LIN {X 39.082,Y -3.308,Z -37.430,A -90.000,B 90.000,C 0.000} C_DIS
LIN {X 39.427,Y -3.308,Z -37.547,A -90.000,B 90.000,C 0.000} C_DIS
LIN {X 39.464,Y -3.308,Z -37.560,A -90.000,B 90.000,C 0.000} C_DIS
LIN {X 41.255,Y -3.308,Z -38.096,A -90.000,B 90.000,C 0.000} C_DIS
LIN {X 41.425,Y -3.308,Z -38.147,A -90.000,B 90.000,C 0.000} C_DIS
LIN {X 41.590,Y -3.308,Z -38.202,A -90.000,B 90.000,C 0.000} C_DIS
LIN {X 41.777,Y -3.308,Z -38.264,A -90.000,B 90.000,C 0.000} C_DIS
LIN {X 42.094,Y -3.308,Z -38.369,A -90.000,B 90.000,C 0.000} C_DIS
LIN {X 42.169,Y -3.308,Z -38.394,A -90.000,B 90.000,C 0.000} C_DIS
LIN {X 42.347,Y -3.308,Z -38.454,A -90.000,B 90.000,C 0.000} C_DIS
LIN {X 42.646,Y -3.308,Z -38.553,A -90.000,B 90.000,C 0.000} C_DIS
LIN {X 43.376,Y -3.308,Z -38.765,A -90.000,B 90.000,C 0.000} C_DIS
LIN {X 43.430,Y -3.308,Z -38.780,A -90.000,B 90.000,C 0.000} C_DIS
LIN {X 43.466,Y -3.308,Z -38.791,A -90.000,B 90.000,C 0.000} C_DIS
LIN {X 43.779,Y -3.308,Z -38.884,A -90.000,B 90.000,C 0.000} C_DIS
LIN {X 43.869,Y -3.308,Z -38.911,A -90.000,B 90.000,C 0.000} C_DIS
LIN {X 43.897,Y -3.308,Z -38.920,A -90.000,B 90.000,C 0.000} C_DIS
LIN {X 44.112,Y -3.308,Z -38.995,A -90.000,B 90.000,C 0.000} C_DIS
LIN {X 45.330,Y -3.308,Z -39.423,A -90.000,B 90.000,C 0.000} C_DIS
LIN {X 46.342,Y -3.308,Z -39.779,A -90.000,B 90.000,C 0.000} C_DIS
LIN {X 46.474,Y -3.308,Z -39.825,A -90.000,B 90.000,C 0.000} C_DIS
LIN {X 46.539,Y -3.308,Z -39.848,A -90.000,B 90.000,C 0.000} C_DIS
LIN {X 46.539,Y -60.000,Z -39.848,A -90.000,B 90.000,C 0.000} C_DIS
LIN {X 103.720,Y -60.000,Z -88.159,A -90.000,B 90.000,C 0.000} C_DIS
LIN {X 103.720,Y -3.308,Z -88.159,A -90.000,B 90.000,C 0.000} C_DIS
LIN {X 103.972,Y -3.308,Z -88.700,A -90.000,B 90.000,C 0.000} C_DIS
LIN {X 104.338,Y -3.308,Z -89.488,A -90.000,B 90.000,C 0.000} C_DIS
LIN {X 104.627,Y -3.308,Z -90.185,A -90.000,B 90.000,C 0.000} C_DIS
LIN {X 104.874,Y -3.308,Z -90.779,A -90.000,B 90.000,C 0.000} C_DIS
LIN {X 104.949,Y -3.308,Z -90.978,A -90.000,B 90.000,C 0.000} C_DIS
LIN {X 105.045,Y -3.308,Z -91.235,A -90.000,B 90.000,C 0.000} C_DIS
LIN {X 105.277,Y -3.308,Z -91.885,A -90.000,B 90.000,C 0.000} C_DIS
LIN {X 105.456,Y -3.308,Z -92.386,A -90.000,B 90.000,C 0.000} C_DIS
LIN {X 105.632,Y -3.308,Z -92.970,A -90.000,B 90.000,C 0.000} C_DIS
LIN {X 105.781,Y -3.308,Z -93.463,A -90.000,B 90.000,C 0.000} C_DIS
LIN {X 105.840,Y -3.308,Z -93.688,A -90.000,B 90.000,C 0.000} C_DIS
LIN {X 105.905,Y -3.308,Z -93.934,A -90.000,B 90.000,C 0.000} C_DIS
LIN {X 106.039,Y -3.308,Z -94.449,A -90.000,B 90.000,C 0.000} C_DIS
LIN {X 106.184,Y -3.308,Z -95.004,A -90.000,B 90.000,C 0.000} C_DIS
LIN {X 106.291,Y -3.308,Z -95.446,A -90.000,B 90.000,C 0.000} C_DIS
LIN {X 106.458,Y -3.308,Z -96.134,A -90.000,B 90.000,C 0.000} C_DIS
LIN {X 106.542,Y -3.308,Z -96.481,A -90.000,B 90.000,C 0.000} C_DIS
LIN {X 106.764,Y -3.308,Z -97.390,A -90.000,B 90.000,C 0.000} C_DIS
LIN {X 106.814,Y -3.308,Z -97.596,A -90.000,B 90.000,C 0.000} C_DIS
LIN {X 107.111,Y -3.308,Z -98.815,A -90.000,B 90.000,C 0.000} C_DIS
LIN {X 107.114,Y -3.308,Z -98.828,A -90.000,B 90.000,C 0.000} C_DIS
LIN {X 107.136,Y -3.308,Z -98.919,A -90.000,B 90.000,C 0.000} C_DIS
LIN {X 107.500,Y -3.308,Z -100.448,A -90.000,B 90.000,C 0.000} C_DIS
LIN {X 107.513,Y -3.308,Z -100.507,A -90.000,B 90.000,C 0.000} C_DIS
LIN {X 107.940,Y -3.308,Z -102.334,A -90.000,B 90.000,C 0.000} C_DIS
LIN {X 108.408,Y -3.308,Z -104.379,A -90.000,B 90.000,C 0.000} C_DIS
LIN {X 108.438,Y -3.308,Z -104.516,A -90.000,B 90.000,C 0.000} C_DIS
LIN {X 108.935,Y -3.308,Z -106.791,A -90.000,B 90.000,C 0.000} C_DIS
LIN {X 108.968,Y -3.308,Z -106.946,A -90.000,B 90.000,C 0.000} C_DIS
LIN {X 109.472,Y -3.308,Z -109.416,A -90.000,B 90.000,C 0.000} C_DIS
LIN {X 109.504,Y -3.308,Z -109.576,A -90.000,B 90.000,C 0.000} C_DIS
LIN {X 109.988,Y -3.308,Z -112.190,A -90.000,B 90.000,C 0.000} C_DIS
LIN {X 110.019,Y -3.308,Z -112.358,A -90.000,B 90.000,C 0.000} C_DIS
LIN {X 110.455,Y -3.308,Z -115.047,A -90.000,B 90.000,C 0.000} C_DIS
LIN {X 110.486,Y -3.308,Z -115.244,A -90.000,B 90.000,C 0.000} C_DIS
LIN {X 110.492,Y -3.308,Z -115.278,A -90.000,B 90.000,C 0.000} C_DIS
LIN {X 110.561,Y -3.308,Z -115.725,A -90.000,B 90.000,C 0.000} C_DIS
LIN {X 110.947,Y -3.308,Z -118.404,A -90.000,B 90.000,C 0.000} C_DIS
LIN {X 110.982,Y -3.308,Z -118.648,A -90.000,B 90.000,C 0.000} C_DIS
LIN {X 111.318,Y -3.308,Z -121.238,A -90.000,B 90.000,C 0.000} C_DIS
LIN {X 111.357,Y -3.308,Z -121.542,A -90.000,B 90.000,C 0.000} C_DIS
LIN {X 111.645,Y -3.308,Z -123.972,A -90.000,B 90.000,C 0.000} C_DIS
LIN {X 111.687,Y -3.308,Z -124.342,A -90.000,B 90.000,C 0.000} C_DIS
LIN {X 111.725,Y -3.308,Z -124.720,A -90.000,B 90.000,C 0.000} C_DIS
LIN {X 111.972,Y -3.308,Z -126.984,A -90.000,B 90.000,C 0.000} C_DIS
LIN {X 112.002,Y -3.308,Z -127.340,A -90.000,B 90.000,C 0.000} C_DIS
LIN {X 112.036,Y -3.308,Z -127.702,A -90.000,B 90.000,C 0.000} C_DIS
LIN {X 112.062,Y -3.308,Z -127.978,A -90.000,B 90.000,C 0.000} C_DIS
LIN {X 112.218,Y -3.308,Z -129.639,A -90.000,B 90.000,C 0.000} C_DIS
LIN {X 112.242,Y -3.308,Z -129.971,A -90.000,B 90.000,C 0.000} C_DIS
LIN {X 112.397,Y -3.308,Z -132.041,A -90.000,B 90.000,C 0.000} C_DIS
LIN {X 112.415,Y -3.308,Z -132.287,A -90.000,B 90.000,C 0.000} C_DIS
LIN {X 112.415,Y -3.308,Z -132.288,A -90.000,B 90.000,C 0.000} C_DIS
LIN {X 112.440,Y -3.308,Z -132.769,A -90.000,B 90.000,C 0.000} C_DIS
LIN {X 112.440,Y -3.308,Z -132.779,A -90.000,B 90.000,C 0.000} C_DIS
LIN {X 112.584,Y -3.308,Z -135.554,A -90.000,B 90.000,C 0.000} C_DIS
LIN {X 112.669,Y -3.308,Z -138.331,A -90.000,B 90.000,C 0.000} C_DIS
LIN {X 112.673,Y -3.308,Z -138.592,A -90.000,B 90.000,C 0.000} C_DIS
LIN {X 112.707,Y -3.308,Z -141.431,A -90.000,B 90.000,C 0.000} C_DIS
LIN {X 112.707,Y -3.308,Z -141.847,A -90.000,B 90.000,C 0.000} C_DIS
LIN {X 112.692,Y -3.308,Z -144.707,A -90.000,B 90.000,C 0.000} C_DIS
LIN {X 112.684,Y -3.308,Z -145.286,A -90.000,B 90.000,C 0.000} C_DIS
LIN {X 112.623,Y -3.308,Z -148.138,A -90.000,B 90.000,C 0.000} C_DIS
LIN {X 112.620,Y -3.308,Z -148.286,A -90.000,B 90.000,C 0.000} C_DIS
LIN {X 112.607,Y -3.308,Z -148.918,A -90.000,B 90.000,C 0.000} C_DIS
LIN {X 112.605,Y -3.308,Z -148.961,A -90.000,B 90.000,C 0.000} C_DIS
LIN {X 112.590,Y -3.308,Z -149.394,A -90.000,B 90.000,C 0.000} C_DIS
LIN {X 112.473,Y -3.308,Z -152.616,A -90.000,B 90.000,C 0.000} C_DIS
LIN {X 112.455,Y -3.308,Z -153.020,A -90.000,B 90.000,C 0.000} C_DIS
LIN {X 112.452,Y -3.308,Z -153.066,A -90.000,B 90.000,C 0.000} C_DIS
LIN {X 112.429,Y -3.308,Z -153.561,A -90.000,B 90.000,C 0.000} C_DIS
LIN {X 112.272,Y -3.308,Z -156.797,A -90.000,B 90.000,C 0.000} C_DIS
LIN {X 112.267,Y -3.308,Z -156.875,A -90.000,B 90.000,C 0.000} C_DIS
LIN {X 112.051,Y -3.308,Z -160.639,A -90.000,B 90.000,C 0.000} C_DIS
LIN {X 112.041,Y -3.308,Z -160.788,A -90.000,B 90.000,C 0.000} C_DIS
LIN {X 111.803,Y -3.308,Z -164.523,A -90.000,B 90.000,C 0.000} C_DIS
LIN {X 111.556,Y -3.308,Z -168.190,A -90.000,B 90.000,C 0.000} C_DIS
LIN {X 111.538,Y -3.308,Z -168.428,A -90.000,B 90.000,C 0.000} C_DIS
LIN {X 111.279,Y -3.308,Z -171.994,A -90.000,B 90.000,C 0.000} C_DIS
LIN {X 111.258,Y -3.308,Z -172.254,A -90.000,B 90.000,C 0.000} C_DIS
LIN {X 110.991,Y -3.308,Z -175.641,A -90.000,B 90.000,C 0.000} C_DIS
LIN {X 110.967,Y -3.308,Z -175.902,A -90.000,B 90.000,C 0.000} C_DIS
LIN {X 110.692,Y -3.308,Z -179.031,A -90.000,B 90.000,C 0.000} C_DIS
LIN {X 110.688,Y -3.308,Z -179.076,A -90.000,B 90.000,C 0.000} C_DIS
LIN {X 110.671,Y -3.308,Z -179.262,A -90.000,B 90.000,C 0.000} C_DIS
LIN {X 110.455,Y -3.308,Z -181.401,A -90.000,B 90.000,C 0.000} C_DIS
LIN {X 110.368,Y -3.308,Z -182.260,A -90.000,B 90.000,C 0.000} C_DIS
LIN {X 110.143,Y -3.308,Z -184.245,A -90.000,B 90.000,C 0.000} C_DIS
LIN {X 110.061,Y -3.308,Z -184.967,A -90.000,B 90.000,C 0.000} C_DIS
LIN {X 109.829,Y -3.308,Z -186.841,A -90.000,B 90.000,C 0.000} C_DIS
LIN {X 109.752,Y -3.308,Z -187.467,A -90.000,B 90.000,C 0.000} C_DIS
LIN {X 109.519,Y -3.308,Z -189.255,A -90.000,B 90.000,C 0.000} C_DIS
LIN {X 109.442,Y -3.308,Z -189.847,A -90.000,B 90.000,C 0.000} C_DIS
LIN {X 109.426,Y -3.308,Z -189.963,A -90.000,B 90.000,C 0.000} C_DIS
LIN {X 109.200,Y -3.308,Z -191.680,A -90.000,B 90.000,C 0.000} C_DIS
LIN {X 109.115,Y -3.308,Z -192.320,A -90.000,B 90.000,C 0.000} C_DIS
LIN {X 108.873,Y -3.308,Z -194.068,A -90.000,B 90.000,C 0.000} C_DIS
LIN {X 108.760,Y -3.308,Z -194.885,A -90.000,B 90.000,C 0.000} C_DIS
LIN {X 108.715,Y -3.308,Z -195.198,A -90.000,B 90.000,C 0.000} C_DIS
LIN {X 108.447,Y -3.308,Z -197.014,A -90.000,B 90.000,C 0.000} C_DIS
LIN {X 108.278,Y -3.308,Z -198.163,A -90.000,B 90.000,C 0.000} C_DIS
LIN {X 107.982,Y -3.308,Z -200.060,A -90.000,B 90.000,C 0.000} C_DIS
LIN {X 107.713,Y -3.308,Z -201.787,A -90.000,B 90.000,C 0.000} C_DIS
LIN {X 107.405,Y -3.308,Z -203.667,A -90.000,B 90.000,C 0.000} C_DIS
LIN {X 106.975,Y -3.308,Z -206.301,A -90.000,B 90.000,C 0.000} C_DIS
LIN {X 106.701,Y -3.308,Z -207.830,A -90.000,B 90.000,C 0.000} C_DIS
LIN {X 106.050,Y -3.308,Z -211.464,A -90.000,B 90.000,C 0.000} C_DIS
LIN {X 105.858,Y -3.308,Z -212.410,A -90.000,B 90.000,C 0.000} C_DIS
LIN {X 104.921,Y -3.308,Z -217.034,A -90.000,B 90.000,C 0.000} C_DIS
LIN {X 104.861,Y -3.308,Z -217.290,A -90.000,B 90.000,C 0.000} C_DIS
LIN {X 104.401,Y -3.308,Z -219.248,A -90.000,B 90.000,C 0.000} C_DIS
LIN {X 103.570,Y -3.308,Z -222.773,A -90.000,B 90.000,C 0.000} C_DIS
LIN {X 103.568,Y -3.308,Z -222.782,A -90.000,B 90.000,C 0.000} C_DIS
LIN {X 103.460,Y -3.308,Z -223.227,A -90.000,B 90.000,C 0.000} C_DIS
LIN {X 103.428,Y -3.308,Z -223.346,A -90.000,B 90.000,C 0.000} C_DIS
LIN {X 101.875,Y -3.308,Z -228.890,A -90.000,B 90.000,C 0.000} C_DIS
LIN {X 101.788,Y -3.308,Z -229.169,A -90.000,B 90.000,C 0.000} C_DIS
LIN {X 100.060,Y -3.308,Z -234.610,A -90.000,B 90.000,C 0.000} C_DIS
LIN {X 99.904,Y -3.308,Z -235.072,A -90.000,B 90.000,C 0.000} C_DIS
LIN {X 99.844,Y -3.308,Z -235.247,A -90.000,B 90.000,C 0.000} C_DIS
LIN {X 99.341,Y -3.308,Z -236.708,A -90.000,B 90.000,C 0.000} C_DIS
LIN {X 98.008,Y -3.308,Z -240.566,A -90.000,B 90.000,C 0.000} C_DIS
LIN {X 97.126,Y -3.308,Z -243.023,A -90.000,B 90.000,C 0.000} C_DIS
LIN {X 96.931,Y -3.308,Z -243.561,A -90.000,B 90.000,C 0.000} C_DIS
LIN {X 96.931,Y -60.000,Z -243.561,A -90.000,B 90.000,C 0.000} C_DIS
LIN {X 103.942,Y -60.000,Z -88.551,A -90.000,B 90.000,C 0.000} C_DIS
LIN {X 103.942,Y -1.308,Z -88.551,A -90.000,B 90.000,C 0.000} C_DIS
LIN {X 104.175,Y -1.308,Z -89.077,A -90.000,B 90.000,C 0.000} C_DIS
LIN {X 104.366,Y -1.308,Z -89.489,A -90.000,B 90.000,C 0.000} C_DIS
LIN {X 104.694,Y -1.308,Z -90.316,A -90.000,B 90.000,C 0.000} C_DIS
LIN {X 104.887,Y -1.308,Z -90.782,A -90.000,B 90.000,C 0.000} C_DIS
LIN {X 105.061,Y -1.308,Z -91.248,A -90.000,B 90.000,C 0.000} C_DIS
LIN {X 105.471,Y -1.308,Z -92.397,A -90.000,B 90.000,C 0.000} C_DIS
LIN {X 105.797,Y -1.308,Z -93.474,A -90.000,B 90.000,C 0.000} C_DIS
LIN {X 106.202,Y -1.308,Z -95.016,A -90.000,B 90.000,C 0.000} C_DIS
LIN {X 106.649,Y -1.308,Z -96.839,A -90.000,B 90.000,C 0.000} C_DIS
LIN {X 107.139,Y -1.308,Z -98.829,A -90.000,B 90.000,C 0.000} C_DIS
LIN {X 107.348,Y -1.308,Z -99.694,A -90.000,B 90.000,C 0.000} C_DIS
LIN {X 107.535,Y -1.308,Z -100.466,A -90.000,B 90.000,C 0.000} C_DIS
LIN {X 107.981,Y -1.308,Z -102.357,A -90.000,B 90.000,C 0.000} C_DIS
LIN {X 108.482,Y -1.308,Z -104.543,A -90.000,B 90.000,C 0.000} C_DIS
LIN {X 108.811,Y -1.308,Z -106.031,A -90.000,B 90.000,C 0.000} C_DIS
LIN {X 109.029,Y -1.308,Z -107.030,A -90.000,B 90.000,C 0.000} C_DIS
LIN {X 109.354,Y -1.308,Z -108.598,A -90.000,B 90.000,C 0.000} C_DIS
LIN {X 109.573,Y -1.308,Z -109.674,A -90.000,B 90.000,C 0.000} C_DIS
LIN {X 109.886,Y -1.308,Z -111.341,A -90.000,B 90.000,C 0.000} C_DIS
LIN {X 110.096,Y -1.308,Z -112.473,A -90.000,B 90.000,C 0.000} C_DIS
LIN {X 110.570,Y -1.308,Z -115.379,A -90.000,B 90.000,C 0.000} C_DIS
LIN {X 110.644,Y -1.308,Z -115.861,A -90.000,B 90.000,C 0.000} C_DIS
LIN {X 111.073,Y -1.308,Z -118.807,A -90.000,B 90.000,C 0.000} C_DIS
LIN {X 111.459,Y -1.308,Z -121.724,A -90.000,B 90.000,C 0.000} C_DIS
LIN {X 111.654,Y -1.308,Z -123.293,A -90.000,B 90.000,C 0.000} C_DIS
LIN {X 111.804,Y -1.308,Z -124.546,A -90.000,B 90.000,C 0.000} C_DIS
LIN {X 111.944,Y -1.308,Z -125.792,A -90.000,B 90.000,C 0.000} C_DIS
LIN {X 112.113,Y -1.308,Z -127.205,A -90.000,B 90.000,C 0.000} C_DIS
LIN {X 112.238,Y -1.308,Z -128.493,A -90.000,B 90.000,C 0.000} C_DIS
LIN {X 112.386,Y -1.308,Z -129.880,A -90.000,B 90.000,C 0.000} C_DIS
LIN {X 112.447,Y -1.308,Z -130.676,A -90.000,B 90.000,C 0.000} C_DIS
LIN {X 112.614,Y -1.308,Z -132.524,A -90.000,B 90.000,C 0.000} C_DIS
LIN {X 112.665,Y -1.308,Z -133.450,A -90.000,B 90.000,C 0.000} C_DIS
LIN {X 112.792,Y -1.308,Z -135.313,A -90.000,B 90.000,C 0.000} C_DIS
LIN {X 112.817,Y -1.308,Z -135.799,A -90.000,B 90.000,C 0.000} C_DIS
LIN {X 112.906,Y -1.308,Z -137.712,A -90.000,B 90.000,C 0.000} C_DIS
LIN {X 112.943,Y -1.308,Z -138.836,A -90.000,B 90.000,C 0.000} C_DIS
LIN {X 112.993,Y -1.308,Z -140.776,A -90.000,B 90.000,C 0.000} C_DIS
LIN {X 113.012,Y -1.308,Z -142.085,A -90.000,B 90.000,C 0.000} C_DIS
LIN {X 113.024,Y -1.308,Z -144.018,A -90.000,B 90.000,C 0.000} C_DIS
LIN {X 113.019,Y -1.308,Z -145.583,A -90.000,B 90.000,C 0.000} C_DIS
LIN {X 112.990,Y -1.308,Z -147.783,A -90.000,B 90.000,C 0.000} C_DIS
LIN {X 112.966,Y -1.308,Z -149.138,A -90.000,B 90.000,C 0.000} C_DIS
LIN {X 112.932,Y -1.308,Z -150.098,A -90.000,B 90.000,C 0.000} C_DIS
LIN {X 112.836,Y -1.308,Z -153.117,A -90.000,B 90.000,C 0.000} C_DIS
LIN {X 112.787,Y -1.308,Z -154.172,A -90.000,B 90.000,C 0.000} C_DIS
LIN {X 112.665,Y -1.308,Z -156.858,A -90.000,B 90.000,C 0.000} C_DIS
LIN {X 112.602,Y -1.308,Z -157.990,A -90.000,B 90.000,C 0.000} C_DIS
LIN {X 112.456,Y -1.308,Z -160.667,A -90.000,B 90.000,C 0.000} C_DIS
LIN {X 112.381,Y -1.308,Z -161.858,A -90.000,B 90.000,C 0.000} C_DIS
LIN {X 112.222,Y -1.308,Z -164.528,A -90.000,B 90.000,C 0.000} C_DIS
LIN {X 112.060,Y -1.308,Z -167.189,A -90.000,B 90.000,C 0.000} C_DIS
LIN {X 111.977,Y -1.308,Z -168.425,A -90.000,B 90.000,C 0.000} C_DIS
LIN {X 111.811,Y -1.308,Z -171.020,A -90.000,B 90.000,C 0.000} C_DIS
LIN {X 111.722,Y -1.308,Z -172.253,A -90.000,B 90.000,C 0.000} C_DIS
LIN {X 111.551,Y -1.308,Z -174.718,A -90.000,B 90.000,C 0.000} C_DIS
LIN {X 111.281,Y -1.308,Z -178.178,A -90.000,B 90.000,C 0.000} C_DIS
LIN {X 111.184,Y -1.308,Z -179.276,A -90.000,B 90.000,C 0.000} C_DIS
LIN {X 111.000,Y -1.308,Z -181.292,A -90.000,B 90.000,C 0.000} C_DIS
LIN {X 110.891,Y -1.308,Z -182.370,A -90.000,B 90.000,C 0.000} C_DIS
LIN {X 110.637,Y -1.308,Z -184.806,A -90.000,B 90.000,C 0.000} C_DIS
LIN {X 110.351,Y -1.308,Z -187.300,A -90.000,B 90.000,C 0.000} C_DIS
LIN {X 110.065,Y -1.308,Z -189.655,A -90.000,B 90.000,C 0.000} C_DIS
LIN {X 110.039,Y -1.308,Z -189.862,A -90.000,B 90.000,C 0.000} C_DIS
LIN {X 109.783,Y -1.308,Z -191.958,A -90.000,B 90.000,C 0.000} C_DIS
LIN {X 109.461,Y -1.308,Z -194.432,A -90.000,B 90.000,C 0.000} C_DIS
LIN {X 108.986,Y -1.308,Z -197.778,A -90.000,B 90.000,C 0.000} C_DIS
LIN {X 108.937,Y -1.308,Z -198.114,A -90.000,B 90.000,C 0.000} C_DIS
LIN {X 108.377,Y -1.308,Z -201.749,A -90.000,B 90.000,C 0.000} C_DIS
LIN {X 107.631,Y -1.308,Z -206.299,A -90.000,B 90.000,C 0.000} C_DIS
LIN {X 107.482,Y -1.308,Z -207.134,A -90.000,B 90.000,C 0.000} C_DIS
LIN {X 106.688,Y -1.308,Z -211.510,A -90.000,B 90.000,C 0.000} C_DIS
LIN {X 106.478,Y -1.308,Z -212.555,A -90.000,B 90.000,C 0.000} C_DIS
LIN {X 105.535,Y -1.308,Z -217.130,A -90.000,B 90.000,C 0.000} C_DIS
LIN {X 105.249,Y -1.308,Z -218.352,A -90.000,B 90.000,C 0.000} C_DIS
LIN {X 104.157,Y -1.308,Z -222.909,A -90.000,B 90.000,C 0.000} C_DIS
LIN {X 104.041,Y -1.308,Z -223.370,A -90.000,B 90.000,C 0.000} C_DIS
LIN {X 103.553,Y -1.308,Z -225.114,A -90.000,B 90.000,C 0.000} C_DIS
LIN {X 103.299,Y -1.308,Z -226.019,A -90.000,B 90.000,C 0.000} C_DIS
LIN {X 102.457,Y -1.308,Z -228.965,A -90.000,B 90.000,C 0.000} C_DIS
LIN {X 101.545,Y -1.308,Z -231.849,A -90.000,B 90.000,C 0.000} C_DIS
LIN {X 100.624,Y -1.308,Z -234.696,A -90.000,B 90.000,C 0.000} C_DIS
LIN {X 100.468,Y -1.308,Z -235.153,A -90.000,B 90.000,C 0.000} C_DIS
LIN {X 99.390,Y -1.308,Z -238.286,A -90.000,B 90.000,C 0.000} C_DIS
LIN {X 98.415,Y -1.308,Z -241.076,A -90.000,B 90.000,C 0.000} C_DIS
LIN {X 97.517,Y -1.308,Z -243.561,A -90.000,B 90.000,C 0.000} C_DIS
LIN {X 97.589,Y -0.997,Z -243.561,A -90.000,B 90.000,C 0.000} C_DIS
LIN {X 97.753,Y -0.254,Z -243.561,A -90.000,B 90.000,C 0.000} C_DIS
LIN {X 97.794,Y -0.012,Z -243.561,A -90.000,B 90.000,C 0.000} C_DIS
LIN {X 98.717,Y -0.012,Z -241.018,A -90.000,B 90.000,C 0.000} C_DIS
LIN {X 100.794,Y -0.012,Z -235.068,A -90.000,B 90.000,C 0.000} C_DIS
LIN {X 100.850,Y -0.012,Z -234.903,A -90.000,B 90.000,C 0.000} C_DIS
LIN {X 102.698,Y -0.012,Z -229.178,A -90.000,B 90.000,C 0.000} C_DIS
LIN {X 104.377,Y -0.012,Z -223.284,A -90.000,B 90.000,C 0.000} C_DIS
LIN {X 104.419,Y -0.012,Z -223.135,A -90.000,B 90.000,C 0.000} C_DIS
LIN {X 105.820,Y -0.012,Z -217.262,A -90.000,B 90.000,C 0.000} C_DIS
LIN {X 106.103,Y -0.012,Z -215.906,A -90.000,B 90.000,C 0.000} C_DIS
LIN {X 107.024,Y -0.012,Z -211.415,A -90.000,B 90.000,C 0.000} C_DIS
LIN {X 107.238,Y -0.012,Z -210.247,A -90.000,B 90.000,C 0.000} C_DIS
LIN {X 107.970,Y -0.012,Z -206.189,A -90.000,B 90.000,C 0.000} C_DIS
LIN {X 108.152,Y -0.012,Z -205.081,A -90.000,B 90.000,C 0.000} C_DIS
LIN {X 108.714,Y -0.012,Z -201.630,A -90.000,B 90.000,C 0.000} C_DIS
LIN {X 109.268,Y -0.012,Z -197.995,A -90.000,B 90.000,C 0.000} C_DIS
LIN {X 109.567,Y -0.012,Z -195.870,A -90.000,B 90.000,C 0.000} C_DIS
LIN {X 109.681,Y -0.012,Z -195.046,A -90.000,B 90.000,C 0.000} C_DIS
LIN {X 109.912,Y -0.012,Z -193.259,A -90.000,B 90.000,C 0.000} C_DIS
LIN {X 110.256,Y -0.012,Z -190.433,A -90.000,B 90.000,C 0.000} C_DIS
LIN {X 110.329,Y -0.012,Z -189.794,A -90.000,B 90.000,C 0.000} C_DIS
LIN {X 110.584,Y -0.012,Z -187.672,A -90.000,B 90.000,C 0.000} C_DIS
LIN {X 110.866,Y -0.012,Z -185.210,A -90.000,B 90.000,C 0.000} C_DIS
LIN {X 111.127,Y -0.012,Z -182.715,A -90.000,B 90.000,C 0.000} C_DIS
LIN {X 111.399,Y -0.012,Z -179.749,A -90.000,B 90.000,C 0.000} C_DIS
LIN {X 111.661,Y -0.012,Z -176.403,A -90.000,B 90.000,C 0.000} C_DIS
LIN {X 111.946,Y -0.012,Z -172.287,A -90.000,B 90.000,C 0.000} C_DIS
LIN {X 112.188,Y -0.012,Z -168.484,A -90.000,B 90.000,C 0.000} C_DIS
LIN {X 112.438,Y -0.012,Z -164.328,A -90.000,B 90.000,C 0.000} C_DIS
LIN {X 112.665,Y -0.012,Z -160.479,A -90.000,B 90.000,C 0.000} C_DIS
LIN {X 112.870,Y -0.012,Z -156.686,A -90.000,B 90.000,C 0.000} C_DIS
LIN {X 113.036,Y -0.012,Z -152.962,A -90.000,B 90.000,C 0.000} C_DIS
LIN {X 113.146,Y -0.012,Z -149.320,A -90.000,B 90.000,C 0.000} C_DIS
LIN {X 113.182,Y -0.012,Z -146.203,A -90.000,B 90.000,C 0.000} C_DIS
LIN {X 113.185,Y -0.012,Z -145.696,A -90.000,B 90.000,C 0.000} C_DIS
LIN {X 113.163,Y -0.012,Z -142.850,A -90.000,B 90.000,C 0.000} C_DIS
LIN {X 113.155,Y -0.012,Z -142.278,A -90.000,B 90.000,C 0.000} C_DIS
LIN {X 113.081,Y -0.012,Z -139.539,A -90.000,B 90.000,C 0.000} C_DIS
LIN {X 113.064,Y -0.012,Z -138.972,A -90.000,B 90.000,C 0.000} C_DIS
LIN {X 112.922,Y -0.012,Z -135.965,A -90.000,B 90.000,C 0.000} C_DIS
LIN {X 112.892,Y -0.012,Z -135.399,A -90.000,B 90.000,C 0.000} C_DIS
LIN {X 112.699,Y -0.012,Z -132.647,A -90.000,B 90.000,C 0.000} C_DIS
LIN {X 112.454,Y -0.012,Z -129.979,A -90.000,B 90.000,C 0.000} C_DIS
LIN {X 112.169,Y -0.012,Z -127.364,A -90.000,B 90.000,C 0.000} C_DIS
LIN {X 111.849,Y -0.012,Z -124.692,A -90.000,B 90.000,C 0.000} C_DIS
LIN {X 111.494,Y -0.012,Z -121.847,A -90.000,B 90.000,C 0.000} C_DIS
LIN {X 111.104,Y -0.012,Z -118.911,A -90.000,B 90.000,C 0.000} C_DIS
LIN {X 110.672,Y -0.012,Z -115.948,A -90.000,B 90.000,C 0.000} C_DIS
LIN {X 110.597,Y -0.012,Z -115.467,A -90.000,B 90.000,C 0.000} C_DIS
LIN {X 110.120,Y -0.012,Z -112.547,A -90.000,B 90.000,C 0.000} C_DIS
LIN {X 109.594,Y -0.012,Z -109.738,A -90.000,B 90.000,C 0.000} C_DIS
LIN {X 109.044,Y -0.012,Z -107.086,A -90.000,B 90.000,C 0.000} C_DIS
LIN {X 108.477,Y -0.012,Z -104.519,A -90.000,B 90.000,C 0.000} C_DIS
LIN {X 107.976,Y -0.012,Z -102.336,A -90.000,B 90.000,C 0.000} C_DIS
LIN {X 107.530,Y -0.012,Z -100.448,A -90.000,B 90.000,C 0.000} C_DIS
LIN {X 107.135,Y -0.012,Z -98.812,A -90.000,B 90.000,C 0.000} C_DIS
LIN {X 106.475,Y -0.012,Z -96.132,A -90.000,B 90.000,C 0.000} C_DIS
LIN {X 106.196,Y -0.012,Z -94.993,A -90.000,B 90.000,C 0.000} C_DIS
LIN {X 105.793,Y -0.012,Z -93.461,A -90.000,B 90.000,C 0.000} C_DIS
LIN {X 105.467,Y -0.012,Z -92.384,A -90.000,B 90.000,C 0.000} C_DIS
LIN {X 105.056,Y -0.012,Z -91.234,A -90.000,B 90.000,C 0.000} C_DIS
LIN {X 104.885,Y -0.012,Z -90.777,A -90.000,B 90.000,C 0.000} C_DIS
LIN {X 104.827,Y -0.012,Z -90.638,A -90.000,B 90.000,C 0.000} C_DIS
LIN {X 104.372,Y -0.012,Z -89.491,A -90.000,B 90.000,C 0.000} C_DIS
LIN {X 104.045,Y -0.012,Z -88.752,A -90.000,B 90.000,C 0.000} C_DIS
LIN {X 104.045,Y -60.000,Z -88.752,A -90.000,B 90.000,C 0.000} C_DIS
LIN {X 43.020,Y -60.000,Z -37.966,A -90.000,B 90.000,C 0.000} C_DIS
LIN {X 43.020,Y -0.012,Z -37.966,A -90.000,B 90.000,C 0.000} C_DIS
LIN {X 42.676,Y -0.012,Z -37.859,A -90.000,B 90.000,C 0.000} C_DIS
LIN {X 39.938,Y -0.012,Z -37.046,A -90.000,B 90.000,C 0.000} C_DIS
LIN {X 39.474,Y -0.012,Z -36.914,A -90.000,B 90.000,C 0.000} C_DIS
LIN {X 38.817,Y -0.012,Z -36.731,A -90.000,B 90.000,C 0.000} C_DIS
LIN {X 36.912,Y -0.012,Z -36.186,A -90.000,B 90.000,C 0.000} C_DIS
LIN {X 36.067,Y -0.012,Z -35.963,A -90.000,B 90.000,C 0.000} C_DIS
LIN {X 34.152,Y -0.012,Z -35.416,A -90.000,B 90.000,C 0.000} C_DIS
LIN {X 32.390,Y -0.012,Z -34.936,A -90.000,B 90.000,C 0.000} C_DIS
LIN {X 32.190,Y -0.012,Z -34.876,A -90.000,B 90.000,C 0.000} C_DIS
LIN {X 30.670,Y -0.012,Z -34.493,A -90.000,B 90.000,C 0.000} C_DIS
LIN {X 30.375,Y -0.012,Z -34.410,A -90.000,B 90.000,C 0.000} C_DIS
LIN {X 29.074,Y -0.012,Z -34.123,A -90.000,B 90.000,C 0.000} C_DIS
LIN {X 28.686,Y -0.012,Z -34.028,A -90.000,B 90.000,C 0.000} C_DIS
LIN {X 28.208,Y -0.012,Z -33.939,A -90.000,B 90.000,C 0.000} C_DIS
LIN {X 27.702,Y -0.012,Z -33.849,A -90.000,B 90.000,C 0.000} C_DIS
LIN {X 26.733,Y -0.012,Z -33.598,A -90.000,B 90.000,C 0.000} C_DIS
LIN {X 25.280,Y -0.012,Z -33.266,A -90.000,B 90.000,C 0.000} C_DIS
LIN {X 23.854,Y -0.012,Z -32.973,A -90.000,B 90.000,C 0.000} C_DIS
LIN {X 20.821,Y -0.012,Z -32.391,A -90.000,B 90.000,C 0.000} C_DIS
LIN {X 19.125,Y -0.012,Z -32.043,A -90.000,B 90.000,C 0.000} C_DIS
LIN {X 15.767,Y -0.012,Z -31.256,A -90.000,B 90.000,C 0.000} C_DIS
LIN {X 14.185,Y -0.012,Z -30.896,A -90.000,B 90.000,C 0.000} C_DIS
LIN {X 12.581,Y -0.012,Z -30.540,A -90.000,B 90.000,C 0.000} C_DIS
LIN {X 10.880,Y -0.012,Z -30.117,A -90.000,B 90.000,C 0.000} C_DIS
LIN {X 8.865,Y -0.012,Z -29.622,A -90.000,B 90.000,C 0.000} C_DIS
LIN {X 3.891,Y -0.012,Z -28.465,A -90.000,B 90.000,C 0.000} C_DIS
LIN {X 1.041,Y -0.012,Z -27.770,A -90.000,B 90.000,C 0.000} C_DIS
LIN {X -1.976,Y -0.012,Z -26.974,A -90.000,B 90.000,C 0.000} C_DIS
LIN {X -4.624,Y -0.012,Z -26.193,A -90.000,B 90.000,C 0.000} C_DIS
LIN {X -7.412,Y -0.012,Z -25.311,A -90.000,B 90.000,C 0.000} C_DIS
LIN {X -7.754,Y -0.012,Z -25.207,A -90.000,B 90.000,C 0.000} C_DIS
LIN {X -10.062,Y -0.012,Z -24.467,A -90.000,B 90.000,C 0.000} C_DIS
LIN {X -10.863,Y -0.012,Z -24.217,A -90.000,B 90.000,C 0.000} C_DIS
LIN {X -13.621,Y -0.012,Z -23.346,A -90.000,B 90.000,C 0.000} C_DIS
LIN {X -13.820,Y -0.012,Z -23.285,A -90.000,B 90.000,C 0.000} C_DIS
LIN {X -16.774,Y -0.012,Z -22.405,A -90.000,B 90.000,C 0.000} C_DIS
LIN {X -16.893,Y -0.012,Z -22.370,A -90.000,B 90.000,C 0.000} C_DIS
LIN {X -17.636,Y -0.012,Z -22.162,A -90.000,B 90.000,C 0.000} C_DIS
LIN {X -19.279,Y -0.012,Z -21.696,A -90.000,B 90.000,C 0.000} C_DIS
LIN {X -21.539,Y -0.012,Z -21.084,A -90.000,B 90.000,C 0.000} C_DIS
LIN {X -26.043,Y -0.012,Z -19.895,A -90.000,B 90.000,C 0.000} C_DIS
LIN {X -26.588,Y -0.012,Z -19.760,A -90.000,B 90.000,C 0.000} C_DIS
LIN {X -28.502,Y -0.012,Z -19.295,A -90.000,B 90.000,C 0.000} C_DIS
LIN {X -31.206,Y -0.012,Z -18.708,A -90.000,B 90.000,C 0.000} C_DIS
LIN {X -33.757,Y -0.012,Z -18.236,A -90.000,B 90.000,C 0.000} C_DIS
LIN {X -34.712,Y -0.012,Z -18.067,A -90.000,B 90.000,C 0.000} C_DIS
LIN {X -37.747,Y -0.012,Z -17.621,A -90.000,B 90.000,C 0.000} C_DIS
LIN {X -38.152,Y -0.012,Z -17.555,A -90.000,B 90.000,C 0.000} C_DIS
LIN {X -40.937,Y -0.012,Z -17.179,A -90.000,B 90.000,C 0.000} C_DIS
LIN {X -41.696,Y -0.012,Z -17.061,A -90.000,B 90.000,C 0.000} C_DIS
LIN {X -42.842,Y -0.012,Z -16.906,A -90.000,B 90.000,C 0.000} C_DIS
LIN {X -45.181,Y -0.012,Z -16.537,A -90.000,B 90.000,C 0.000} C_DIS
LIN {X -45.737,Y -0.012,Z -16.454,A -90.000,B 90.000,C 0.000} C_DIS
LIN {X -48.058,Y -0.012,Z -16.058,A -90.000,B 90.000,C 0.000} C_DIS
LIN {X -49.516,Y -0.012,Z -15.762,A -90.000,B 90.000,C 0.000} C_DIS
LIN {X -50.309,Y -0.012,Z -15.602,A -90.000,B 90.000,C 0.000} C_DIS
LIN {X -52.298,Y -0.012,Z -15.130,A -90.000,B 90.000,C 0.000} C_DIS
LIN {X -53.891,Y -0.012,Z -14.701,A -90.000,B 90.000,C 0.000} C_DIS
LIN {X -55.198,Y -0.012,Z -14.324,A -90.000,B 90.000,C 0.000} C_DIS
LIN {X -56.332,Y -0.012,Z -14.007,A -90.000,B 90.000,C 0.000} C_DIS
LIN {X -57.641,Y -0.012,Z -13.652,A -90.000,B 90.000,C 0.000} C_DIS
LIN {X -59.127,Y -0.012,Z -13.251,A -90.000,B 90.000,C 0.000} C_DIS
LIN {X -60.166,Y -0.012,Z -12.960,A -90.000,B 90.000,C 0.000} C_DIS
LIN {X -61.184,Y -0.012,Z -12.702,A -90.000,B 90.000,C 0.000} C_DIS
LIN {X -62.291,Y -0.012,Z -12.477,A -90.000,B 90.000,C 0.000} C_DIS
LIN {X -62.770,Y -0.012,Z -12.387,A -90.000,B 90.000,C 0.000} C_DIS
LIN {X -63.035,Y -0.012,Z -12.350,A -90.000,B 90.000,C 0.000} C_DIS
LIN {X -64.074,Y -0.012,Z -12.192,A -90.000,B 90.000,C 0.000} C_DIS
LIN {X -64.556,Y -0.012,Z -12.151,A -90.000,B 90.000,C 0.000} C_DIS
LIN {X -65.927,Y -0.012,Z -12.042,A -90.000,B 90.000,C 0.000} C_DIS
LIN {X -67.369,Y -0.012,Z -11.981,A -90.000,B 90.000,C 0.000} C_DIS
LIN {X -68.812,Y -0.012,Z -11.939,A -90.000,B 90.000,C 0.000} C_DIS
LIN {X -70.189,Y -0.012,Z -11.883,A -90.000,B 90.000,C 0.000} C_DIS
LIN {X -71.023,Y -0.012,Z -11.818,A -90.000,B 90.000,C 0.000} C_DIS
LIN {X -72.129,Y -0.012,Z -11.687,A -90.000,B 90.000,C 0.000} C_DIS
LIN {X -73.241,Y -0.012,Z -11.518,A -90.000,B 90.000,C 0.000} C_DIS
LIN {X -74.294,Y -0.012,Z -11.380,A -90.000,B 90.000,C 0.000} C_DIS
LIN {X -74.779,Y -0.012,Z -11.338,A -90.000,B 90.000,C 0.000} C_DIS
LIN {X -75.788,Y -0.012,Z -11.262,A -90.000,B 90.000,C 0.000} C_DIS
LIN {X -76.595,Y -0.012,Z -11.236,A -90.000,B 90.000,C 0.000} C_DIS
LIN {X -76.881,Y -0.012,Z -11.223,A -90.000,B 90.000,C 0.000} C_DIS
LIN {X -77.658,Y -0.012,Z -11.218,A -90.000,B 90.000,C 0.000} C_DIS
LIN {X -77.953,Y -0.012,Z -11.212,A -90.000,B 90.000,C 0.000} C_DIS
LIN {X -78.827,Y -0.012,Z -11.211,A -90.000,B 90.000,C 0.000} C_DIS
LIN {X -79.219,Y -0.012,Z -11.205,A -90.000,B 90.000,C 0.000} C_DIS
LIN {X -80.206,Y -0.012,Z -11.169,A -90.000,B 90.000,C 0.000} C_DIS
LIN {X -80.638,Y -0.012,Z -11.166,A -90.000,B 90.000,C 0.000} C_DIS
LIN {X -81.548,Y -0.012,Z -11.134,A -90.000,B 90.000,C 0.000} C_DIS
LIN {X -82.119,Y -0.012,Z -11.133,A -90.000,B 90.000,C 0.000} C_DIS
LIN {X -82.935,Y -0.012,Z -11.120,A -90.000,B 90.000,C 0.000} C_DIS
LIN {X -83.757,Y -0.012,Z -11.111,A -90.000,B 90.000,C 0.000} C_DIS
LIN {X -85.248,Y -0.012,Z -11.141,A -90.000,B 90.000,C 0.000} C_DIS
LIN {X -85.753,Y -0.012,Z -11.159,A -90.000,B 90.000,C 0.000} C_DIS
LIN {X -87.138,Y -0.012,Z -11.278,A -90.000,B 90.000,C 0.000} C_DIS
LIN {X -87.533,Y -0.012,Z -11.333,A -90.000,B 90.000,C 0.000} C_DIS
LIN {X -88.765,Y -0.012,Z -11.522,A -90.000,B 90.000,C 0.000} C_DIS
LIN {X -88.932,Y -0.012,Z -11.549,A -90.000,B 90.000,C 0.000} C_DIS
LIN {X -90.192,Y -0.012,Z -11.831,A -90.000,B 90.000,C 0.000} C_DIS
LIN {X -90.405,Y -0.012,Z -11.883,A -90.000,B 90.000,C 0.000} C_DIS
LIN {X -90.656,Y -0.012,Z -11.951,A -90.000,B 90.000,C 0.000} C_DIS
LIN {X -91.880,Y -0.012,Z -12.313,A -90.000,B 90.000,C 0.000} C_DIS
LIN {X -93.124,Y -0.012,Z -12.761,A -90.000,B 90.000,C 0.000} C_DIS
LIN {X -93.538,Y -0.012,Z -12.922,A -90.000,B 90.000,C 0.000} C_DIS
LIN {X -93.992,Y -0.012,Z -13.111,A -90.000,B 90.000,C 0.000} C_DIS
LIN {X -94.547,Y -0.012,Z -13.336,A -90.000,B 90.000,C 0.000} C_DIS
LIN {X -94.813,Y -0.012,Z -13.457,A -90.000,B 90.000,C 0.000} C_DIS
LIN {X -95.652,Y -0.012,Z -13.832,A -90.000,B 90.000,C 0.000} C_DIS
LIN {X -96.130,Y -0.012,Z -14.062,A -90.000,B 90.000,C 0.000} C_DIS
LIN {X -97.061,Y -0.012,Z -14.512,A -90.000,B 90.000,C 0.000} C_DIS
LIN {X -98.451,Y -0.012,Z -15.222,A -90.000,B 90.000,C 0.000} C_DIS
LIN {X -99.427,Y -0.012,Z -15.739,A -90.000,B 90.000,C 0.000} C_DIS
LIN {X -100.226,Y -0.012,Z -16.182,A -90.000,B 90.000,C 0.000} C_DIS
LIN {X -100.368,Y -0.012,Z -16.265,A -90.000,B 90.000,C 0.000} C_DIS
LIN {X -100.488,Y -0.012,Z -16.339,A -90.000,B 90.000,C 0.000} C_DIS
LIN {X -100.938,Y -0.012,Z -16.608,A -90.000,B 90.000,C 0.000} C_DIS
LIN {X -101.304,Y -0.012,Z -16.834,A -90.000,B 90.000,C 0.000} C_DIS
LIN {X -101.747,Y -0.012,Z -17.127,A -90.000,B 90.000,C 0.000} C_DIS
LIN {X -102.089,Y -0.012,Z -17.376,A -90.000,B 90.000,C 0.000} C_DIS
LIN {X -102.470,Y -0.012,Z -17.669,A -90.000,B 90.000,C 0.000} C_DIS
LIN {X -102.769,Y -0.012,Z -17.907,A -90.000,B 90.000,C 0.000} C_DIS
LIN {X -103.064,Y -0.012,Z -18.156,A -90.000,B 90.000,C 0.000} C_DIS
LIN {X -103.290,Y -0.012,Z -18.344,A -90.000,B 90.000,C 0.000} C_DIS
LIN {X -103.372,Y -0.012,Z -18.397,A -90.000,B 90.000,C 0.000} C_DIS
LIN {X -103.540,Y -0.012,Z -18.488,A -90.000,B 90.000,C 0.000} C_DIS
LIN {X -103.696,Y -0.012,Z -18.560,A -90.000,B 90.000,C 0.000} C_DIS
LIN {X -104.031,Y -0.012,Z -18.692,A -90.000,B 90.000,C 0.000} C_DIS
LIN {X -104.302,Y -0.012,Z -18.784,A -90.000,B 90.000,C 0.000} C_DIS
LIN {X -104.361,Y -0.012,Z -18.803,A -90.000,B 90.000,C 0.000} C_DIS
LIN {X -104.830,Y -0.012,Z -18.935,A -90.000,B 90.000,C 0.000} C_DIS
LIN {X -105.040,Y -0.012,Z -18.987,A -90.000,B 90.000,C 0.000} C_DIS
LIN {X -105.840,Y -0.012,Z -19.168,A -90.000,B 90.000,C 0.000} C_DIS
LIN {X -106.017,Y -0.012,Z -19.204,A -90.000,B 90.000,C 0.000} C_DIS
LIN {X -106.783,Y -0.012,Z -19.379,A -90.000,B 90.000,C 0.000} C_DIS
LIN {X -107.114,Y -0.012,Z -19.458,A -90.000,B 90.000,C 0.000} C_DIS
LIN {X -107.732,Y -0.012,Z -19.621,A -90.000,B 90.000,C 0.000} C_DIS
LIN {X -108.330,Y -0.012,Z -19.805,A -90.000,B 90.000,C 0.000} C_DIS
LIN {X -108.791,Y -0.012,Z -19.963,A -90.000,B 90.000,C 0.000} C_DIS
LIN {X -109.029,Y -0.012,Z -20.051,A -90.000,B 90.000,C 0.000} C_DIS
LIN {X -109.357,Y -0.012,Z -20.175,A -90.000,B 90.000,C 0.000} C_DIS
LIN {X -109.798,Y -0.012,Z -20.379,A -90.000,B 90.000,C 0.000} C_DIS
LIN {X -109.978,Y -0.012,Z -20.465,A -90.000,B 90.000,C 0.000} C_DIS
LIN {X -110.319,Y -0.012,Z -20.622,A -90.000,B 90.000,C 0.000} C_DIS
LIN {X -110.590,Y -0.012,Z -20.783,A -90.000,B 90.000,C 0.000} C_DIS
LIN {X -110.798,Y -0.012,Z -20.898,A -90.000,B 90.000,C 0.000} C_DIS
LIN {X -111.216,Y -0.012,Z -21.146,A -90.000,B 90.000,C 0.000} C_DIS
LIN {X -111.461,Y -0.012,Z -21.322,A -90.000,B 90.000,C 0.000} C_DIS
LIN {X -111.658,Y -0.012,Z -21.455,A -90.000,B 90.000,C 0.000} C_DIS
LIN {X -112.049,Y -0.012,Z -21.745,A -90.000,B 90.000,C 0.000} C_DIS
LIN {X -112.268,Y -0.012,Z -21.933,A -90.000,B 90.000,C 0.000} C_DIS
LIN {X -112.459,Y -0.012,Z -22.088,A -90.000,B 90.000,C 0.000} C_DIS
LIN {X -112.818,Y -0.012,Z -22.417,A -90.000,B 90.000,C 0.000} C_DIS
LIN {X -113.198,Y -0.012,Z -22.795,A -90.000,B 90.000,C 0.000} C_DIS
LIN {X -113.522,Y -0.012,Z -23.158,A -90.000,B 90.000,C 0.000} C_DIS
LIN {X -113.873,Y -0.012,Z -23.571,A -90.000,B 90.000,C 0.000} C_DIS
LIN {X -114.477,Y -0.012,Z -24.411,A -90.000,B 90.000,C 0.000} C_DIS
LIN {X -114.765,Y -0.012,Z -24.887,A -90.000,B 90.000,C 0.000} C_DIS
LIN {X -115.008,Y -0.012,Z -25.309,A -90.000,B 90.000,C 0.000} C_DIS
LIN {X -115.177,Y -0.012,Z -25.638,A -90.000,B 90.000,C 0.000} C_DIS
LIN {X -115.264,Y -0.012,Z -25.815,A -90.000,B 90.000,C 0.000} C_DIS
LIN {X -115.431,Y -0.012,Z -26.168,A -90.000,B 90.000,C 0.000} C_DIS
LIN {X -115.513,Y -0.012,Z -26.351,A -90.000,B 90.000,C 0.000} C_DIS
LIN {X -115.732,Y -0.012,Z -26.810,A -90.000,B 90.000,C 0.000} C_DIS
LIN {X -115.830,Y -0.012,Z -26.994,A -90.000,B 90.000,C 0.000} C_DIS
LIN {X -115.864,Y -0.012,Z -27.045,A -90.000,B 90.000,C 0.000} C_DIS
LIN {X -116.050,Y -0.012,Z -27.265,A -90.000,B 90.000,C 0.000} C_DIS
LIN {X -116.446,Y -0.012,Z -27.703,A -90.000,B 90.000,C 0.000} C_DIS
LIN {X -116.650,Y -0.012,Z -27.954,A -90.000,B 90.000,C 0.000} C_DIS
LIN {X -117.116,Y -0.012,Z -28.594,A -90.000,B 90.000,C 0.000} C_DIS
LIN {X -117.273,Y -0.012,Z -28.837,A -90.000,B 90.000,C 0.000} C_DIS
LIN {X -117.417,Y -0.012,Z -29.080,A -90.000,B 90.000,C 0.000} C_DIS
LIN {X -117.663,Y -0.012,Z -29.500,A -90.000,B 90.000,C 0.000} C_DIS
LIN {X -117.799,Y -0.012,Z -29.743,A -90.000,B 90.000,C 0.000} C_DIS
LIN {X -117.924,Y -0.012,Z -29.988,A -90.000,B 90.000,C 0.000} C_DIS
LIN {X -118.246,Y -0.012,Z -30.696,A -90.000,B 90.000,C 0.000} C_DIS
LIN {X -118.346,Y -0.012,Z -30.950,A -90.000,B 90.000,C 0.000} C_DIS
LIN {X -118.501,Y -0.012,Z -31.413,A -90.000,B 90.000,C 0.000} C_DIS
LIN {X -118.585,Y -0.012,Z -31.674,A -90.000,B 90.000,C 0.000} C_DIS
LIN {X -118.650,Y -0.012,Z -31.942,A -90.000,B 90.000,C 0.000} C_DIS
LIN {X -118.757,Y -0.012,Z -32.418,A -90.000,B 90.000,C 0.000} C_DIS
LIN {X -118.802,Y -0.012,Z -32.688,A -90.000,B 90.000,C 0.000} C_DIS
LIN {X -118.860,Y -0.012,Z -33.172,A -90.000,B 90.000,C 0.000} C_DIS
LIN {X -118.881,Y -0.012,Z -33.443,A -90.000,B 90.000,C 0.000} C_DIS
LIN {X -118.889,Y -0.012,Z -33.931,A -90.000,B 90.000,C 0.000} C_DIS
LIN {X -118.885,Y -0.012,Z -34.199,A -90.000,B 90.000,C 0.000} C_DIS
LIN {X -118.839,Y -0.012,Z -34.711,A -90.000,B 90.000,C 0.000} C_DIS
LIN {X -118.804,Y -0.012,Z -34.981,A -90.000,B 90.000,C 0.000} C_DIS
LIN {X -118.714,Y -0.012,Z -35.455,A -90.000,B 90.000,C 0.000} C_DIS
LIN {X -118.640,Y -0.012,Z -35.763,A -90.000,B 90.000,C 0.000} C_DIS
LIN {X -118.500,Y -0.012,Z -36.231,A -90.000,B 90.000,C 0.000} C_DIS
LIN {X -118.465,Y -0.012,Z -36.337,A -90.000,B 90.000,C 0.000} C_DIS
LIN {X -118.563,Y -0.012,Z -36.490,A -90.000,B 90.000,C 0.000} C_DIS
LIN {X -118.795,Y -0.012,Z -36.914,A -90.000,B 90.000,C 0.000} C_DIS
LIN {X -118.974,Y -0.012,Z -37.298,A -90.000,B 90.000,C 0.000} C_DIS
LIN {X -119.161,Y -0.012,Z -37.743,A -90.000,B 90.000,C 0.000} C_DIS
LIN {X -119.300,Y -0.012,Z -38.205,A -90.000,B 90.000,C 0.000} C_DIS
LIN {X -119.342,Y -0.012,Z -38.349,A -90.000,B 90.000,C 0.000} C_DIS
LIN {X -119.412,Y -0.012,Z -38.572,A -90.000,B 90.000,C 0.000} C_DIS
LIN {X -119.515,Y -0.012,Z -39.048,A -90.000,B 90.000,C 0.000} C_DIS
LIN {X -119.536,Y -0.012,Z -39.193,A -90.000,B 90.000,C 0.000} C_DIS
LIN {X -119.584,Y -0.012,Z -39.481,A -90.000,B 90.000,C 0.000} C_DIS
LIN {X -119.638,Y -0.012,Z -39.965,A -90.000,B 90.000,C 0.000} C_DIS
LIN {X -119.643,Y -0.012,Z -40.127,A -90.000,B 90.000,C 0.000} C_DIS
LIN {X -119.656,Y -0.012,Z -40.422,A -90.000,B 90.000,C 0.000} C_DIS
LIN {X -119.659,Y -0.012,Z -40.908,A -90.000,B 90.000,C 0.000} C_DIS
LIN {X -119.630,Y -0.012,Z -41.387,A -90.000,B 90.000,C 0.000} C_DIS
LIN {X -119.584,Y -0.012,Z -41.871,A -90.000,B 90.000,C 0.000} C_DIS
LIN {X -119.507,Y -0.012,Z -42.409,A -90.000,B 90.000,C 0.000} C_DIS
LIN {X -119.414,Y -0.012,Z -42.887,A -90.000,B 90.000,C 0.000} C_DIS
LIN {X -119.309,Y -0.012,Z -43.408,A -90.000,B 90.000,C 0.000} C_DIS
LIN {X -119.178,Y -0.012,Z -43.941,A -90.000,B 90.000,C 0.000} C_DIS
LIN {X -119.010,Y -0.012,Z -44.559,A -90.000,B 90.000,C 0.000} C_DIS
LIN {X -118.883,Y -0.012,Z -45.012,A -90.000,B 90.000,C 0.000} C_DIS
LIN {X -118.851,Y -0.012,Z -45.146,A -90.000,B 90.000,C 0.000} C_DIS
LIN {X -119.044,Y -0.012,Z -46.324,A -90.000,B 90.000,C 0.000} C_DIS
LIN {X -119.098,Y -0.012,Z -46.814,A -90.000,B 90.000,C 0.000} C_DIS
LIN {X -119.164,Y -0.012,Z -47.798,A -90.000,B 90.000,C 0.000} C_DIS
LIN {X -119.168,Y -0.012,Z -48.271,A -90.000,B 90.000,C 0.000} C_DIS
LIN {X -119.071,Y -0.012,Z -49.446,A -90.000,B 90.000,C 0.000} C_DIS
LIN {X -119.029,Y -0.012,Z -49.894,A -90.000,B 90.000,C 0.000} C_DIS
LIN {X -118.933,Y -0.012,Z -50.371,A -90.000,B 90.000,C 0.000} C_DIS
LIN {X -118.589,Y -0.012,Z -51.702,A -90.000,B 90.000,C 0.000} C_DIS
LIN {X -118.444,Y -0.012,Z -52.173,A -90.000,B 90.000,C 0.000} C_DIS
LIN {X -117.916,Y -0.012,Z -53.679,A -90.000,B 90.000,C 0.000} C_DIS
LIN {X -117.265,Y -0.012,Z -55.362,A -90.000,B 90.000,C 0.000} C_DIS
LIN {X -116.560,Y -0.012,Z -57.201,A -90.000,B 90.000,C 0.000} C_DIS
LIN {X -115.877,Y -0.012,Z -59.154,A -90.000,B 90.000,C 0.000} C_DIS
LIN {X -115.192,Y -0.012,Z -61.162,A -90.000,B 90.000,C 0.000} C_DIS
LIN {X -114.504,Y -0.012,Z -63.106,A -90.000,B 90.000,C 0.000} C_DIS
LIN {X -113.804,Y -0.012,Z -64.883,A -90.000,B 90.000,C 0.000} C_DIS
LIN {X -113.616,Y -0.012,Z -65.333,A -90.000,B 90.000,C 0.000} C_DIS
LIN {X -112.896,Y -0.012,Z -66.840,A -90.000,B 90.000,C 0.000} C_DIS
LIN {X -112.695,Y -0.012,Z -67.210,A -90.000,B 90.000,C 0.000} C_DIS
LIN {X -112.624,Y -0.012,Z -67.334,A -90.000,B 90.000,C 0.000} C_DIS
LIN {X -112.269,Y -0.012,Z -67.929,A -90.000,B 90.000,C 0.000} C_DIS
LIN {X -111.819,Y -0.012,Z -68.679,A -90.000,B 90.000,C 0.000} C_DIS
LIN {X -111.541,Y -0.012,Z -69.078,A -90.000,B 90.000,C 0.000} C_DIS
LIN {X -111.083,Y -0.012,Z -69.701,A -90.000,B 90.000,C 0.000} C_DIS
LIN {X -110.606,Y -0.012,Z -70.334,A -90.000,B 90.000,C 0.000} C_DIS
LIN {X -110.288,Y -0.012,Z -70.702,A -90.000,B 90.000,C 0.000} C_DIS
LIN {X -109.667,Y -0.012,Z -71.415,A -90.000,B 90.000,C 0.000} C_DIS
LIN {X -109.172,Y -0.012,Z -71.959,A -90.000,B 90.000,C 0.000} C_DIS
LIN {X -109.035,Y -0.012,Z -72.093,A -90.000,B 90.000,C 0.000} C_DIS
LIN {X -107.723,Y -0.012,Z -73.434,A -90.000,B 90.000,C 0.000} C_DIS
LIN {X -107.627,Y -0.012,Z -73.525,A -90.000,B 90.000,C 0.000} C_DIS
LIN {X -106.394,Y -0.012,Z -74.617,A -90.000,B 90.000,C 0.000} C_DIS
LIN {X -106.187,Y -0.012,Z -74.811,A -90.000,B 90.000,C 0.000} C_DIS
LIN {X -105.826,Y -0.012,Z -75.131,A -90.000,B 90.000,C 0.000} C_DIS
LIN {X -104.651,Y -0.012,Z -75.989,A -90.000,B 90.000,C 0.000} C_DIS
LIN {X -104.225,Y -0.012,Z -76.315,A -90.000,B 90.000,C 0.000} C_DIS
LIN {X -103.908,Y -0.012,Z -76.543,A -90.000,B 90.000,C 0.000} C_DIS
LIN {X -103.832,Y -0.012,Z -76.596,A -90.000,B 90.000,C 0.000} C_DIS
LIN {X -103.584,Y -0.012,Z -76.743,A -90.000,B 90.000,C 0.000} C_DIS
LIN {X -103.178,Y -0.012,Z -76.962,A -90.000,B 90.000,C 0.000} C_DIS
LIN {X -101.934,Y -0.012,Z -77.644,A -90.000,B 90.000,C 0.000} C_DIS
LIN {X -101.598,Y -0.012,Z -77.812,A -90.000,B 90.000,C 0.000} C_DIS
LIN {X -101.508,Y -0.012,Z -77.856,A -90.000,B 90.000,C 0.000} C_DIS
LIN {X -101.061,Y -0.012,Z -78.022,A -90.000,B 90.000,C 0.000} C_DIS
LIN {X -99.978,Y -0.012,Z -78.324,A -90.000,B 90.000,C 0.000} C_DIS
LIN {X -99.201,Y -0.012,Z -78.553,A -90.000,B 90.000,C 0.000} C_DIS
LIN {X -98.729,Y -0.012,Z -78.653,A -90.000,B 90.000,C 0.000} C_DIS
LIN {X -98.249,Y -0.012,Z -78.703,A -90.000,B 90.000,C 0.000} C_DIS
LIN {X -97.762,Y -0.012,Z -78.746,A -90.000,B 90.000,C 0.000} C_DIS
LIN {X -97.113,Y -0.012,Z -78.822,A -90.000,B 90.000,C 0.000} C_DIS
LIN {X -96.633,Y -0.012,Z -78.872,A -90.000,B 90.000,C 0.000} C_DIS
LIN {X -96.150,Y -0.012,Z -78.872,A -90.000,B 90.000,C 0.000} C_DIS
LIN {X -95.684,Y -0.012,Z -78.857,A -90.000,B 90.000,C 0.000} C_DIS
LIN {X -94.785,Y -0.012,Z -78.855,A -90.000,B 90.000,C 0.000} C_DIS
LIN {X -94.622,Y -0.012,Z -78.847,A -90.000,B 90.000,C 0.000} C_DIS
LIN {X -94.457,Y -0.012,Z -78.835,A -90.000,B 90.000,C 0.000} C_DIS
LIN {X -93.389,Y -0.012,Z -78.769,A -90.000,B 90.000,C 0.000} C_DIS
LIN {X -92.204,Y -0.012,Z -78.711,A -90.000,B 90.000,C 0.000} C_DIS
LIN {X -91.267,Y -0.012,Z -78.692,A -90.000,B 90.000,C 0.000} C_DIS
LIN {X -90.741,Y -0.012,Z -78.712,A -90.000,B 90.000,C 0.000} C_DIS
LIN {X -90.566,Y -0.012,Z -78.735,A -90.000,B 90.000,C 0.000} C_DIS
LIN {X -90.481,Y -0.012,Z -78.784,A -90.000,B 90.000,C 0.000} C_DIS
LIN {X -89.739,Y -0.012,Z -79.295,A -90.000,B 90.000,C 0.000} C_DIS
LIN {X -89.343,Y -0.012,Z -79.572,A -90.000,B 90.000,C 0.000} C_DIS
LIN {X -89.110,Y -0.012,Z -79.729,A -90.000,B 90.000,C 0.000} C_DIS
LIN {X -88.672,Y -0.012,Z -80.032,A -90.000,B 90.000,C 0.000} C_DIS
LIN {X -88.403,Y -0.012,Z -80.206,A -90.000,B 90.000,C 0.000} C_DIS
LIN {X -87.937,Y -0.012,Z -80.517,A -90.000,B 90.000,C 0.000} C_DIS
LIN {X -87.632,Y -0.012,Z -80.702,A -90.000,B 90.000,C 0.000} C_DIS
LIN {X -87.141,Y -0.012,Z -81.009,A -90.000,B 90.000,C 0.000} C_DIS
LIN {X -86.457,Y -0.012,Z -81.404,A -90.000,B 90.000,C 0.000} C_DIS
LIN {X -85.266,Y -0.012,Z -82.084,A -90.000,B 90.000,C 0.000} C_DIS
LIN {X -84.476,Y -0.012,Z -82.559,A -90.000,B 90.000,C 0.000} C_DIS
LIN {X -83.599,Y -0.012,Z -83.137,A -90.000,B 90.000,C 0.000} C_DIS
LIN {X -82.563,Y -0.012,Z -83.907,A -90.000,B 90.000,C 0.000} C_DIS
LIN {X -81.361,Y -0.012,Z -84.829,A -90.000,B 90.000,C 0.000} C_DIS
LIN {X -80.009,Y -0.012,Z -85.843,A -90.000,B 90.000,C 0.000} C_DIS
LIN {X -78.415,Y -0.012,Z -86.965,A -90.000,B 90.000,C 0.000} C_DIS
LIN {X -76.522,Y -0.012,Z -88.187,A -90.000,B 90.000,C 0.000} C_DIS
LIN {X -74.424,Y -0.012,Z -89.516,A -90.000,B 90.000,C 0.000} C_DIS
LIN {X -72.195,Y -0.012,Z -90.967,A -90.000,B 90.000,C 0.000} C_DIS
LIN {X -69.928,Y -0.012,Z -92.539,A -90.000,B 90.000,C 0.000} C_DIS
LIN {X -68.045,Y -0.012,Z -93.981,A -90.000,B 90.000,C 0.000} C_DIS
LIN {X -66.968,Y -0.012,Z -94.883,A -90.000,B 90.000,C 0.000} C_DIS
LIN {X -65.752,Y -0.012,Z -95.904,A -90.000,B 90.000,C 0.000} C_DIS
LIN {X -64.591,Y -0.012,Z -96.959,A -90.000,B 90.000,C 0.000} C_DIS
LIN {X -63.592,Y -0.012,Z -97.869,A -90.000,B 90.000,C 0.000} C_DIS
LIN {X -61.369,Y -0.012,Z -100.044,A -90.000,B 90.000,C 0.000} C_DIS
LIN {X -58.886,Y -0.012,Z -102.631,A -90.000,B 90.000,C 0.000} C_DIS
LIN {X -56.407,Y -0.012,Z -105.317,A -90.000,B 90.000,C 0.000} C_DIS
LIN {X -55.979,Y -0.012,Z -105.789,A -90.000,B 90.000,C 0.000} C_DIS
LIN {X -54.001,Y -0.012,Z -107.989,A -90.000,B 90.000,C 0.000} C_DIS
LIN {X -52.956,Y -0.012,Z -109.162,A -90.000,B 90.000,C 0.000} C_DIS
LIN {X -51.776,Y -0.012,Z -110.527,A -90.000,B 90.000,C 0.000} C_DIS
LIN {X -51.593,Y -0.012,Z -110.734,A -90.000,B 90.000,C 0.000} C_DIS
LIN {X -50.908,Y -0.012,Z -111.532,A -90.000,B 90.000,C 0.000} C_DIS
LIN {X -50.615,Y -0.012,Z -111.882,A -90.000,B 90.000,C 0.000} C_DIS
LIN {X -50.071,Y -0.012,Z -112.549,A -90.000,B 90.000,C 0.000} C_DIS
LIN {X -48.076,Y -0.012,Z -115.001,A -90.000,B 90.000,C 0.000} C_DIS
LIN {X -46.330,Y -0.012,Z -117.187,A -90.000,B 90.000,C 0.000} C_DIS
LIN {X -45.900,Y -0.012,Z -117.749,A -90.000,B 90.000,C 0.000} C_DIS
LIN {X -45.900,Y -60.000,Z -117.749,A -90.000,B 90.000,C 0.000} C_DIS
LIN {X -36.524,Y -60.000,Z -136.225,A -90.000,B 90.000,C 0.000} C_DIS
LIN {X -36.524,Y -0.012,Z -136.225,A -90.000,B 90.000,C 0.000} C_DIS
LIN {X -36.254,Y -0.012,Z -136.761,A -90.000,B 90.000,C 0.000} C_DIS
LIN {X -36.207,Y -0.012,Z -136.854,A -90.000,B 90.000,C 0.000} C_DIS
LIN {X -35.975,Y -0.012,Z -137.283,A -90.000,B 90.000,C 0.000} C_DIS
LIN {X -33.459,Y -0.012,Z -141.487,A -90.000,B 90.000,C 0.000} C_DIS
LIN {X -33.184,Y -0.012,Z -141.890,A -90.000,B 90.000,C 0.000} C_DIS
LIN {X -30.243,Y -0.012,Z -145.784,A -90.000,B 90.000,C 0.000} C_DIS
LIN {X -29.928,Y -0.012,Z -146.157,A -90.000,B 90.000,C 0.000} C_DIS
LIN {X -27.159,Y -0.012,Z -149.340,A -90.000,B 90.000,C 0.000} C_DIS
LIN {X -26.867,Y -0.012,Z -149.676,A -90.000,B 90.000,C 0.000} C_DIS
LIN {X -23.872,Y -0.012,Z -152.884,A -90.000,B 90.000,C 0.000} C_DIS
LIN {X -21.568,Y -0.012,Z -155.370,A -90.000,B 90.000,C 0.000} C_DIS
LIN {X -20.070,Y -0.012,Z -157.233,A -90.000,B 90.000,C 0.000} C_DIS
LIN {X -19.177,Y -0.012,Z -158.579,A -90.000,B 90.000,C 0.000} C_DIS
LIN {X -18.638,Y -0.012,Z -159.619,A -90.000,B 90.000,C 0.000} C_DIS
LIN {X -18.290,Y -0.012,Z -160.493,A -90.000,B 90.000,C 0.000} C_DIS
LIN {X -17.986,Y -0.012,Z -161.354,A -90.000,B 90.000,C 0.000} C_DIS
LIN {X -17.900,Y -0.012,Z -161.759,A -90.000,B 90.000,C 0.000} C_DIS
LIN {X -17.892,Y -0.012,Z -162.216,A -90.000,B 90.000,C 0.000} C_DIS
LIN {X -18.036,Y -0.012,Z -163.102,A -90.000,B 90.000,C 0.000} C_DIS
LIN {X -18.496,Y -0.012,Z -164.611,A -90.000,B 90.000,C 0.000} C_DIS
LIN {X -19.296,Y -0.012,Z -166.630,A -90.000,B 90.000,C 0.000} C_DIS
LIN {X -20.261,Y -0.012,Z -168.672,A -90.000,B 90.000,C 0.000} C_DIS
LIN {X -21.395,Y -0.012,Z -170.734,A -90.000,B 90.000,C 0.000} C_DIS
LIN {X -22.601,Y -0.012,Z -172.604,A -90.000,B 90.000,C 0.000} C_DIS
LIN {X -23.910,Y -0.012,Z -174.320,A -90.000,B 90.000,C 0.000} C_DIS
LIN {X -25.346,Y -0.012,Z -175.927,A -90.000,B 90.000,C 0.000} C_DIS
LIN {X -27.245,Y -0.012,Z -177.784,A -90.000,B 90.000,C 0.000} C_DIS
LIN {X -29.319,Y -0.012,Z -179.606,A -90.000,B 90.000,C 0.000} C_DIS
LIN {X -31.978,Y -0.012,Z -181.764,A -90.000,B 90.000,C 0.000} C_DIS
LIN {X -34.890,Y -0.012,Z -183.987,A -90.000,B 90.000,C 0.000} C_DIS
LIN {X -37.766,Y -0.012,Z -186.085,A -90.000,B 90.000,C 0.000} C_DIS
LIN {X -41.248,Y -0.012,Z -188.538,A -90.000,B 90.000,C 0.000} C_DIS
LIN {X -45.242,Y -0.012,Z -191.208,A -90.000,B 90.000,C 0.000} C_DIS
LIN {X -50.006,Y -0.012,Z -194.210,A -90.000,B 90.000,C 0.000} C_DIS
LIN {X -55.525,Y -0.012,Z -197.499,A -90.000,B 90.000,C 0.000} C_DIS
LIN {X -57.173,Y -0.012,Z -198.433,A -90.000,B 90.000,C 0.000} C_DIS
LIN {X -62.455,Y -0.012,Z -201.433,A -90.000,B 90.000,C 0.000} C_DIS
LIN {X -63.977,Y -0.012,Z -202.283,A -90.000,B 90.000,C 0.000} C_DIS
LIN {X -70.430,Y -0.012,Z -205.898,A -90.000,B 90.000,C 0.000} C_DIS
LIN {X -78.914,Y -0.012,Z -210.687,A -90.000,B 90.000,C 0.000} C_DIS
LIN {X -87.582,Y -0.012,Z -215.715,A -90.000,B 90.000,C 0.000} C_DIS
LIN {X -87.946,Y -0.012,Z -215.930,A -90.000,B 90.000,C 0.000} C_DIS
LIN {X -96.289,Y -0.012,Z -221.004,A -90.000,B 90.000,C 0.000} C_DIS
LIN {X -104.356,Y -0.012,Z -226.087,A -90.000,B 90.000,C 0.000} C_DIS
LIN {X -112.131,Y -0.012,Z -231.111,A -90.000,B 90.000,C 0.000} C_DIS
LIN {X -120.015,Y -0.013,Z -236.267,A -90.000,B 90.000,C 0.000} C_DIS
LIN {X -120.015,Y -1.308,Z -236.441,A -90.000,B 90.000,C 0.000} C_DIS
LIN {X -112.041,Y -1.308,Z -231.229,A -90.000,B 90.000,C 0.000} C_DIS
LIN {X -104.272,Y -1.308,Z -226.213,A -90.000,B 90.000,C 0.000} C_DIS
LIN {X -96.221,Y -1.308,Z -221.133,A -90.000,B 90.000,C 0.000} C_DIS
LIN {X -87.897,Y -1.308,Z -216.055,A -90.000,B 90.000,C 0.000} C_DIS
LIN {X -87.478,Y -1.308,Z -215.807,A -90.000,B 90.000,C 0.000} C_DIS
LIN {X -84.198,Y -1.308,Z -213.890,A -90.000,B 90.000,C 0.000} C_DIS
LIN {X -78.887,Y -1.308,Z -210.799,A -90.000,B 90.000,C 0.000} C_DIS
LIN {X -76.503,Y -1.308,Z -209.441,A -90.000,B 90.000,C 0.000} C_DIS
LIN {X -68.941,Y -1.308,Z -205.159,A -90.000,B 90.000,C 0.000} C_DIS
LIN {X -62.448,Y -1.308,Z -201.511,A -90.000,B 90.000,C 0.000} C_DIS
LIN {X -61.742,Y -1.308,Z -201.106,A -90.000,B 90.000,C 0.000} C_DIS
LIN {X -55.455,Y -1.308,Z -197.526,A -90.000,B 90.000,C 0.000} C_DIS
LIN {X -50.004,Y -1.308,Z -194.270,A -90.000,B 90.000,C 0.000} C_DIS
LIN {X -45.238,Y -1.308,Z -191.264,A -90.000,B 90.000,C 0.000} C_DIS
LIN {X -41.243,Y -1.308,Z -188.593,A -90.000,B 90.000,C 0.000} C_DIS
LIN {X -37.762,Y -1.308,Z -186.140,A -90.000,B 90.000,C 0.000} C_DIS
LIN {X -34.792,Y -1.308,Z -183.976,A -90.000,B 90.000,C 0.000} C_DIS
LIN {X -31.974,Y -1.308,Z -181.825,A -90.000,B 90.000,C 0.000} C_DIS
LIN {X -29.316,Y -1.308,Z -179.669,A -90.000,B 90.000,C 0.000} C_DIS
LIN {X -27.196,Y -1.308,Z -177.807,A -90.000,B 90.000,C 0.000} C_DIS
LIN {X -25.312,Y -1.308,Z -175.966,A -90.000,B 90.000,C 0.000} C_DIS
LIN {X -23.882,Y -1.308,Z -174.367,A -90.000,B 90.000,C 0.000} C_DIS
LIN {X -22.544,Y -1.308,Z -172.615,A -90.000,B 90.000,C 0.000} C_DIS
LIN {X -21.319,Y -1.308,Z -170.723,A -90.000,B 90.000,C 0.000} C_DIS
LIN {X -20.211,Y -1.308,Z -168.717,A -90.000,B 90.000,C 0.000} C_DIS
LIN {X -19.202,Y -1.308,Z -166.595,A -90.000,B 90.000,C 0.000} C_DIS
LIN {X -18.402,Y -1.308,Z -164.593,A -90.000,B 90.000,C 0.000} C_DIS
LIN {X -17.945,Y -1.308,Z -163.104,A -90.000,B 90.000,C 0.000} C_DIS
LIN {X -17.797,Y -1.308,Z -162.201,A -90.000,B 90.000,C 0.000} C_DIS
LIN {X -17.805,Y -1.308,Z -161.742,A -90.000,B 90.000,C 0.000} C_DIS
LIN {X -17.887,Y -1.308,Z -161.357,A -90.000,B 90.000,C 0.000} C_DIS
LIN {X -18.189,Y -1.308,Z -160.497,A -90.000,B 90.000,C 0.000} C_DIS
LIN {X -18.323,Y -1.308,Z -160.174,A -90.000,B 90.000,C 0.000} C_DIS
LIN {X -18.555,Y -1.308,Z -159.591,A -90.000,B 90.000,C 0.000} C_DIS
LIN {X -18.752,Y -1.308,Z -159.219,A -90.000,B 90.000,C 0.000} C_DIS
LIN {X -19.096,Y -1.308,Z -158.551,A -90.000,B 90.000,C 0.000} C_DIS
LIN {X -19.424,Y -1.308,Z -158.066,A -90.000,B 90.000,C 0.000} C_DIS
LIN {X -19.999,Y -1.308,Z -157.197,A -90.000,B 90.000,C 0.000} C_DIS
LIN {X -20.525,Y -1.308,Z -156.551,A -90.000,B 90.000,C 0.000} C_DIS
LIN {X -21.510,Y -1.308,Z -155.326,A -90.000,B 90.000,C 0.000} C_DIS
LIN {X -22.266,Y -1.308,Z -154.515,A -90.000,B 90.000,C 0.000} C_DIS
LIN {X -23.839,Y -1.308,Z -152.818,A -90.000,B 90.000,C 0.000} C_DIS
LIN {X -25.382,Y -1.308,Z -151.174,A -90.000,B 90.000,C 0.000} C_DIS
LIN {X -26.802,Y -1.308,Z -149.654,A -90.000,B 90.000,C 0.000} C_DIS
LIN {X -28.532,Y -1.308,Z -147.677,A -90.000,B 90.000,C 0.000} C_DIS
LIN {X -29.879,Y -1.308,Z -146.128,A -90.000,B 90.000,C 0.000} C_DIS
LIN {X -30.199,Y -1.308,Z -145.748,A -90.000,B 90.000,C 0.000} C_DIS
LIN {X -31.729,Y -1.308,Z -143.739,A -90.000,B 90.000,C 0.000} C_DIS
LIN {X -33.142,Y -1.308,Z -141.868,A -90.000,B 90.000,C 0.000} C_DIS
LIN {X -33.426,Y -1.308,Z -141.449,A -90.000,B 90.000,C 0.000} C_DIS
LIN {X -34.766,Y -1.308,Z -139.236,A -90.000,B 90.000,C 0.000} C_DIS
LIN {X -35.942,Y -1.308,Z -137.271,A -90.000,B 90.000,C 0.000} C_DIS
LIN {X -36.194,Y -1.308,Z -136.803,A -90.000,B 90.000,C 0.000} C_DIS
LIN {X -36.410,Y -1.308,Z -136.379,A -90.000,B 90.000,C 0.000} C_DIS
LIN {X -36.410,Y -60.000,Z -136.379,A -90.000,B 90.000,C 0.000} C_DIS
LIN {X -45.193,Y -60.000,Z -118.671,A -90.000,B 90.000,C 0.000} C_DIS
LIN {X -45.193,Y -1.308,Z -118.671,A -90.000,B 90.000,C 0.000} C_DIS
LIN {X -46.341,Y -1.308,Z -117.173,A -90.000,B 90.000,C 0.000} C_DIS
LIN {X -48.091,Y -1.308,Z -114.983,A -90.000,B 90.000,C 0.000} C_DIS
LIN {X -50.089,Y -1.308,Z -112.526,A -90.000,B 90.000,C 0.000} C_DIS
LIN {X -50.815,Y -1.308,Z -111.639,A -90.000,B 90.000,C 0.000} C_DIS
LIN {X -53.730,Y -1.308,Z -108.162,A -90.000,B 90.000,C 0.000} C_DIS
LIN {X -54.391,Y -1.308,Z -107.398,A -90.000,B 90.000,C 0.000} C_DIS
LIN {X -55.024,Y -1.308,Z -106.657,A -90.000,B 90.000,C 0.000} C_DIS
LIN {X -56.869,Y -1.308,Z -104.572,A -90.000,B 90.000,C 0.000} C_DIS
LIN {X -58.953,Y -1.308,Z -102.282,A -90.000,B 90.000,C 0.000} C_DIS
LIN {X -60.350,Y -1.308,Z -100.815,A -90.000,B 90.000,C 0.000} C_DIS
LIN {X -61.318,Y -1.308,Z -99.808,A -90.000,B 90.000,C 0.000} C_DIS
LIN {X -63.727,Y -1.308,Z -97.456,A -90.000,B 90.000,C 0.000} C_DIS
LIN {X -65.103,Y -1.308,Z -96.217,A -90.000,B 90.000,C 0.000} C_DIS
LIN {X -65.803,Y -1.308,Z -95.581,A -90.000,B 90.000,C 0.000} C_DIS
LIN {X -67.011,Y -1.308,Z -94.583,A -90.000,B 90.000,C 0.000} C_DIS
LIN {X -67.995,Y -1.308,Z -93.760,A -90.000,B 90.000,C 0.000} C_DIS
LIN {X -69.101,Y -1.308,Z -92.927,A -90.000,B 90.000,C 0.000} C_DIS
LIN {X -70.106,Y -1.308,Z -92.159,A -90.000,B 90.000,C 0.000} C_DIS
LIN {X -72.112,Y -1.308,Z -90.775,A -90.000,B 90.000,C 0.000} C_DIS
LIN {X -73.216,Y -1.308,Z -90.062,A -90.000,B 90.000,C 0.000} C_DIS
LIN {X -74.304,Y -1.308,Z -89.354,A -90.000,B 90.000,C 0.000} C_DIS
LIN {X -75.607,Y -1.308,Z -88.530,A -90.000,B 90.000,C 0.000} C_DIS
LIN {X -76.373,Y -1.308,Z -88.048,A -90.000,B 90.000,C 0.000} C_DIS
LIN {X -78.244,Y -1.308,Z -86.843,A -90.000,B 90.000,C 0.000} C_DIS
LIN {X -79.908,Y -1.308,Z -85.674,A -90.000,B 90.000,C 0.000} C_DIS
LIN {X -80.223,Y -1.308,Z -85.448,A -90.000,B 90.000,C 0.000} C_DIS
LIN {X -81.576,Y -1.308,Z -84.433,A -90.000,B 90.000,C 0.000} C_DIS
LIN {X -82.758,Y -1.308,Z -83.522,A -90.000,B 90.000,C 0.000} C_DIS
LIN {X -83.605,Y -1.308,Z -82.886,A -90.000,B 90.000,C 0.000} C_DIS
LIN {X -84.140,Y -1.308,Z -82.526,A -90.000,B 90.000,C 0.000} C_DIS
LIN {X -84.458,Y -1.308,Z -82.305,A -90.000,B 90.000,C 0.000} C_DIS
LIN {X -85.116,Y -1.308,Z -81.897,A -90.000,B 90.000,C 0.000} C_DIS
LIN {X -85.423,Y -1.308,Z -81.697,A -90.000,B 90.000,C 0.000} C_DIS
LIN {X -86.044,Y -1.308,Z -81.328,A -90.000,B 90.000,C 0.000} C_DIS
LIN {X -86.175,Y -1.308,Z -81.245,A -90.000,B 90.000,C 0.000} C_DIS
LIN {X -87.006,Y -1.308,Z -80.744,A -90.000,B 90.000,C 0.000} C_DIS
LIN {X -87.233,Y -1.308,Z -80.600,A -90.000,B 90.000,C 0.000} C_DIS
LIN {X -88.016,Y -1.308,Z -80.088,A -90.000,B 90.000,C 0.000} C_DIS
LIN {X -88.778,Y -1.308,Z -79.564,A -90.000,B 90.000,C 0.000} C_DIS
LIN {X -89.434,Y -1.308,Z -79.102,A -90.000,B 90.000,C 0.000} C_DIS
LIN {X -90.030,Y -1.308,Z -78.685,A -90.000,B 90.000,C 0.000} C_DIS
LIN {X -90.275,Y -1.308,Z -78.522,A -90.000,B 90.000,C 0.000} C_DIS
LIN {X -90.337,Y -1.308,Z -78.489,A -90.000,B 90.000,C 0.000} C_DIS
LIN {X -90.503,Y -1.308,Z -78.478,A -90.000,B 90.000,C 0.000} C_DIS
LIN {X -90.635,Y -1.308,Z -78.466,A -90.000,B 90.000,C 0.000} C_DIS
LIN {X -91.141,Y -1.308,Z -78.466,A -90.000,B 90.000,C 0.000} C_DIS
LIN {X -92.222,Y -1.308,Z -78.504,A -90.000,B 90.000,C 0.000} C_DIS
LIN {X -92.809,Y -1.308,Z -78.533,A -90.000,B 90.000,C 0.000} C_DIS
LIN {X -93.301,Y -1.308,Z -78.551,A -90.000,B 90.000,C 0.000} C_DIS
LIN {X -94.402,Y -1.308,Z -78.584,A -90.000,B 90.000,C 0.000} C_DIS
LIN {X -94.640,Y -1.308,Z -78.599,A -90.000,B 90.000,C 0.000} C_DIS
LIN {X -95.122,Y -1.308,Z -78.599,A -90.000,B 90.000,C 0.000} C_DIS
LIN {X -96.038,Y -1.308,Z -78.566,A -90.000,B 90.000,C 0.000} C_DIS
LIN {X -96.314,Y -1.308,Z -78.567,A -90.000,B 90.000,C 0.000} C_DIS
LIN {X -96.594,Y -1.308,Z -78.560,A -90.000,B 90.000,C 0.000} C_DIS
LIN {X -96.790,Y -1.308,Z -78.548,A -90.000,B 90.000,C 0.000} C_DIS
LIN {X -97.074,Y -1.308,Z -78.510,A -90.000,B 90.000,C 0.000} C_DIS
LIN {X -97.482,Y -1.308,Z -78.448,A -90.000,B 90.000,C 0.000} C_DIS
LIN {X -98.376,Y -1.308,Z -78.342,A -90.000,B 90.000,C 0.000} C_DIS
LIN {X -98.848,Y -1.308,Z -78.272,A -90.000,B 90.000,C 0.000} C_DIS
LIN {X -99.309,Y -1.308,Z -78.154,A -90.000,B 90.000,C 0.000} C_DIS
LIN {X -99.892,Y -1.308,Z -77.967,A -90.000,B 90.000,C 0.000} C_DIS
LIN {X -100.949,Y -1.308,Z -77.652,A -90.000,B 90.000,C 0.000} C_DIS
LIN {X -101.395,Y -1.308,Z -77.486,A -90.000,B 90.000,C 0.000} C_DIS
LIN {X -101.822,Y -1.308,Z -77.274,A -90.000,B 90.000,C 0.000} C_DIS
LIN {X -102.773,Y -1.308,Z -76.756,A -90.000,B 90.000,C 0.000} C_DIS
LIN {X -103.481,Y -1.308,Z -76.377,A -90.000,B 90.000,C 0.000} C_DIS
LIN {X -103.883,Y -1.308,Z -76.122,A -90.000,B 90.000,C 0.000} C_DIS
LIN {X -104.701,Y -1.308,Z -75.519,A -90.000,B 90.000,C 0.000} C_DIS
LIN {X -105.503,Y -1.308,Z -74.957,A -90.000,B 90.000,C 0.000} C_DIS
LIN {X -105.749,Y -1.308,Z -74.766,A -90.000,B 90.000,C 0.000} C_DIS
LIN {X -105.875,Y -1.308,Z -74.660,A -90.000,B 90.000,C 0.000} C_DIS
LIN {X -105.962,Y -1.308,Z -74.583,A -90.000,B 90.000,C 0.000} C_DIS
LIN {X -107.298,Y -1.308,Z -73.460,A -90.000,B 90.000,C 0.000} C_DIS
LIN {X -107.611,Y -1.308,Z -73.183,A -90.000,B 90.000,C 0.000} C_DIS
LIN {X -108.817,Y -1.308,Z -72.006,A -90.000,B 90.000,C 0.000} C_DIS
LIN {X -109.006,Y -1.308,Z -71.832,A -90.000,B 90.000,C 0.000} C_DIS
LIN {X -109.260,Y -1.308,Z -71.559,A -90.000,B 90.000,C 0.000} C_DIS
LIN {X -109.529,Y -1.308,Z -71.265,A -90.000,B 90.000,C 0.000} C_DIS
LIN {X -110.452,Y -1.308,Z -70.243,A -90.000,B 90.000,C 0.000} C_DIS
LIN {X -110.703,Y -1.308,Z -69.914,A -90.000,B 90.000,C 0.000} C_DIS
LIN {X -111.594,Y -1.308,Z -68.723,A -90.000,B 90.000,C 0.000} C_DIS
LIN {X -111.669,Y -1.308,Z -68.620,A -90.000,B 90.000,C 0.000} C_DIS
LIN {X -111.786,Y -1.308,Z -68.441,A -90.000,B 90.000,C 0.000} C_DIS
LIN {X -112.575,Y -1.308,Z -67.129,A -90.000,B 90.000,C 0.000} C_DIS
LIN {X -112.811,Y -1.308,Z -66.703,A -90.000,B 90.000,C 0.000} C_DIS
LIN {X -113.520,Y -1.308,Z -65.215,A -90.000,B 90.000,C 0.000} C_DIS
LIN {X -113.711,Y -1.308,Z -64.767,A -90.000,B 90.000,C 0.000} C_DIS
LIN {X -114.400,Y -1.308,Z -63.018,A -90.000,B 90.000,C 0.000} C_DIS
LIN {X -115.095,Y -1.308,Z -61.050,A -90.000,B 90.000,C 0.000} C_DIS
LIN {X -115.747,Y -1.308,Z -59.135,A -90.000,B 90.000,C 0.000} C_DIS
LIN {X -116.417,Y -1.308,Z -57.213,A -90.000,B 90.000,C 0.000} C_DIS
LIN {X -117.095,Y -1.308,Z -55.436,A -90.000,B 90.000,C 0.000} C_DIS
LIN {X -117.720,Y -1.308,Z -53.814,A -90.000,B 90.000,C 0.000} C_DIS
LIN {X -118.229,Y -1.308,Z -52.355,A -90.000,B 90.000,C 0.000} C_DIS
LIN {X -118.327,Y -1.308,Z -52.064,A -90.000,B 90.000,C 0.000} C_DIS
LIN {X -118.380,Y -1.308,Z -51.895,A -90.000,B 90.000,C 0.000} C_DIS
LIN {X -118.713,Y -1.308,Z -50.609,A -90.000,B 90.000,C 0.000} C_DIS
LIN {X -118.797,Y -1.308,Z -50.240,A -90.000,B 90.000,C 0.000} C_DIS
LIN {X -118.818,Y -1.308,Z -50.137,A -90.000,B 90.000,C 0.000} C_DIS
LIN {X -118.863,Y -1.308,Z -49.761,A -90.000,B 90.000,C 0.000} C_DIS
LIN {X -118.968,Y -1.308,Z -48.553,A -90.000,B 90.000,C 0.000} C_DIS
LIN {X -118.975,Y -1.308,Z -48.072,A -90.000,B 90.000,C 0.000} C_DIS
LIN {X -118.915,Y -1.308,Z -47.120,A -90.000,B 90.000,C 0.000} C_DIS
LIN {X -118.873,Y -1.308,Z -46.640,A -90.000,B 90.000,C 0.000} C_DIS
LIN {X -118.673,Y -1.308,Z -45.365,A -90.000,B 90.000,C 0.000} C_DIS
LIN {X -118.684,Y -1.308,Z -45.313,A -90.000,B 90.000,C 0.000} C_DIS
LIN {X -118.973,Y -1.308,Z -44.237,A -90.000,B 90.000,C 0.000} C_DIS
LIN {X -119.106,Y -1.308,Z -43.696,A -90.000,B 90.000,C 0.000} C_DIS
LIN {X -119.155,Y -1.308,Z -43.481,A -90.000,B 90.000,C 0.000} C_DIS
LIN {X -119.317,Y -1.308,Z -42.692,A -90.000,B 90.000,C 0.000} C_DIS
LIN {X -119.390,Y -1.308,Z -42.178,A -90.000,B 90.000,C 0.000} C_DIS
LIN {X -119.420,Y -1.308,Z -41.929,A -90.000,B 90.000,C 0.000} C_DIS
LIN {X -119.442,Y -1.308,Z -41.697,A -90.000,B 90.000,C 0.000} C_DIS
LIN {X -119.467,Y -1.308,Z -41.206,A -90.000,B 90.000,C 0.000} C_DIS
LIN {X -119.474,Y -1.308,Z -40.722,A -90.000,B 90.000,C 0.000} C_DIS
LIN {X -119.450,Y -1.308,Z -40.259,A -90.000,B 90.000,C 0.000} C_DIS
LIN {X -119.408,Y -1.308,Z -39.779,A -90.000,B 90.000,C 0.000} C_DIS
LIN {X -119.331,Y -1.308,Z -39.344,A -90.000,B 90.000,C 0.000} C_DIS
LIN {X -119.261,Y -1.308,Z -38.979,A -90.000,B 90.000,C 0.000} C_DIS
LIN {X -119.240,Y -1.308,Z -38.870,A -90.000,B 90.000,C 0.000} C_DIS
LIN {X -119.101,Y -1.308,Z -38.408,A -90.000,B 90.000,C 0.000} C_DIS
LIN {X -118.969,Y -1.308,Z -38.003,A -90.000,B 90.000,C 0.000} C_DIS
LIN {X -118.826,Y -1.308,Z -37.650,A -90.000,B 90.000,C 0.000} C_DIS
LIN {X -118.768,Y -1.308,Z -37.530,A -90.000,B 90.000,C 0.000} C_DIS
LIN {X -118.426,Y -1.308,Z -36.848,A -90.000,B 90.000,C 0.000} C_DIS
LIN {X -118.318,Y -1.308,Z -36.680,A -90.000,B 90.000,C 0.000} C_DIS
LIN {X -118.406,Y -1.308,Z -36.403,A -90.000,B 90.000,C 0.000} C_DIS
LIN {X -118.546,Y -1.308,Z -35.936,A -90.000,B 90.000,C 0.000} C_DIS
LIN {X -118.622,Y -1.308,Z -35.607,A -90.000,B 90.000,C 0.000} C_DIS
LIN {X -118.733,Y -1.308,Z -35.046,A -90.000,B 90.000,C 0.000} C_DIS
LIN {X -118.769,Y -1.308,Z -34.765,A -90.000,B 90.000,C 0.000} C_DIS
LIN {X -118.815,Y -1.308,Z -34.281,A -90.000,B 90.000,C 0.000} C_DIS
LIN {X -118.819,Y -1.308,Z -34.011,A -90.000,B 90.000,C 0.000} C_DIS
LIN {X -118.815,Y -1.308,Z -33.524,A -90.000,B 90.000,C 0.000} C_DIS
LIN {X -118.795,Y -1.308,Z -33.252,A -90.000,B 90.000,C 0.000} C_DIS
LIN {X -118.741,Y -1.308,Z -32.768,A -90.000,B 90.000,C 0.000} C_DIS
LIN {X -118.698,Y -1.308,Z -32.496,A -90.000,B 90.000,C 0.000} C_DIS
LIN {X -118.594,Y -1.308,Z -32.020,A -90.000,B 90.000,C 0.000} C_DIS
LIN {X -118.530,Y -1.308,Z -31.751,A -90.000,B 90.000,C 0.000} C_DIS
LIN {X -118.448,Y -1.308,Z -31.487,A -90.000,B 90.000,C 0.000} C_DIS
LIN {X -118.297,Y -1.308,Z -31.024,A -90.000,B 90.000,C 0.000} C_DIS
LIN {X -118.199,Y -1.308,Z -30.768,A -90.000,B 90.000,C 0.000} C_DIS
LIN {X -117.888,Y -1.308,Z -30.073,A -90.000,B 90.000,C 0.000} C_DIS
LIN {X -117.764,Y -1.308,Z -29.827,A -90.000,B 90.000,C 0.000} C_DIS
LIN {X -117.630,Y -1.308,Z -29.583,A -90.000,B 90.000,C 0.000} C_DIS
LIN {X -117.325,Y -1.308,Z -29.055,A -90.000,B 90.000,C 0.000} C_DIS
LIN {X -117.245,Y -1.308,Z -28.918,A -90.000,B 90.000,C 0.000} C_DIS
LIN {X -117.089,Y -1.308,Z -28.674,A -90.000,B 90.000,C 0.000} C_DIS
LIN {X -116.628,Y -1.308,Z -28.034,A -90.000,B 90.000,C 0.000} C_DIS
LIN {X -116.525,Y -1.308,Z -27.907,A -90.000,B 90.000,C 0.000} C_DIS
LIN {X -116.425,Y -1.308,Z -27.787,A -90.000,B 90.000,C 0.000} C_DIS
LIN {X -116.101,Y -1.308,Z -27.423,A -90.000,B 90.000,C 0.000} C_DIS
LIN {X -115.990,Y -1.308,Z -27.308,A -90.000,B 90.000,C 0.000} C_DIS
LIN {X -115.866,Y -1.308,Z -27.172,A -90.000,B 90.000,C 0.000} C_DIS
LIN {X -115.735,Y -1.308,Z -27.038,A -90.000,B 90.000,C 0.000} C_DIS
LIN {X -115.670,Y -1.308,Z -26.960,A -90.000,B 90.000,C 0.000} C_DIS
LIN {X -115.618,Y -1.308,Z -26.870,A -90.000,B 90.000,C 0.000} C_DIS
LIN {X -115.530,Y -1.308,Z -26.698,A -90.000,B 90.000,C 0.000} C_DIS
LIN {X -115.317,Y -1.308,Z -26.277,A -90.000,B 90.000,C 0.000} C_DIS
LIN {X -115.176,Y -1.308,Z -25.997,A -90.000,B 90.000,C 0.000} C_DIS
LIN {X -114.906,Y -1.308,Z -25.491,A -90.000,B 90.000,C 0.000} C_DIS
LIN {X -114.801,Y -1.308,Z -25.299,A -90.000,B 90.000,C 0.000} C_DIS
LIN {X -114.669,Y -1.308,Z -25.069,A -90.000,B 90.000,C 0.000} C_DIS
LIN {X -114.394,Y -1.308,Z -24.619,A -90.000,B 90.000,C 0.000} C_DIS
LIN {X -114.120,Y -1.308,Z -24.221,A -90.000,B 90.000,C 0.000} C_DIS
LIN {X -113.800,Y -1.308,Z -23.771,A -90.000,B 90.000,C 0.000} C_DIS
LIN {X -113.448,Y -1.308,Z -23.354,A -90.000,B 90.000,C 0.000} C_DIS
LIN {X -113.134,Y -1.308,Z -22.987,A -90.000,B 90.000,C 0.000} C_DIS
LIN {X -112.749,Y -1.308,Z -22.607,A -90.000,B 90.000,C 0.000} C_DIS
LIN {X -112.399,Y -1.308,Z -22.275,A -90.000,B 90.000,C 0.000} C_DIS
LIN {X -112.176,Y -1.308,Z -22.097,A -90.000,B 90.000,C 0.000} C_DIS
LIN {X -111.980,Y -1.308,Z -21.936,A -90.000,B 90.000,C 0.000} C_DIS
LIN {X -111.597,Y -1.308,Z -21.641,A -90.000,B 90.000,C 0.000} C_DIS
LIN {X -111.358,Y -1.308,Z -21.488,A -90.000,B 90.000,C 0.000} C_DIS
LIN {X -111.140,Y -1.308,Z -21.340,A -90.000,B 90.000,C 0.000} C_DIS
LIN {X -110.729,Y -1.308,Z -21.086,A -90.000,B 90.000,C 0.000} C_DIS
LIN {X -110.470,Y -1.308,Z -20.950,A -90.000,B 90.000,C 0.000} C_DIS
LIN {X -110.232,Y -1.308,Z -20.818,A -90.000,B 90.000,C 0.000} C_DIS
LIN {X -109.797,Y -1.308,Z -20.609,A -90.000,B 90.000,C 0.000} C_DIS
LIN {X -109.512,Y -1.308,Z -20.486,A -90.000,B 90.000,C 0.000} C_DIS
LIN {X -109.257,Y -1.308,Z -20.370,A -90.000,B 90.000,C 0.000} C_DIS
LIN {X -108.531,Y -1.308,Z -20.107,A -90.000,B 90.000,C 0.000} C_DIS
LIN {X -108.217,Y -1.308,Z -19.995,A -90.000,B 90.000,C 0.000} C_DIS
LIN {X -107.598,Y -1.308,Z -19.808,A -90.000,B 90.000,C 0.000} C_DIS
LIN {X -106.960,Y -1.308,Z -19.645,A -90.000,B 90.000,C 0.000} C_DIS
LIN {X -106.491,Y -1.308,Z -19.529,A -90.000,B 90.000,C 0.000} C_DIS
LIN {X -106.261,Y -1.308,Z -19.478,A -90.000,B 90.000,C 0.000} C_DIS
LIN {X -105.847,Y -1.308,Z -19.391,A -90.000,B 90.000,C 0.000} C_DIS
LIN {X -105.372,Y -1.308,Z -19.310,A -90.000,B 90.000,C 0.000} C_DIS
LIN {X -105.210,Y -1.308,Z -19.278,A -90.000,B 90.000,C 0.000} C_DIS
LIN {X -104.686,Y -1.308,Z -19.195,A -90.000,B 90.000,C 0.000} C_DIS
LIN {X -104.515,Y -1.308,Z -19.164,A -90.000,B 90.000,C 0.000} C_DIS
LIN {X -104.132,Y -1.308,Z -19.085,A -90.000,B 90.000,C 0.000} C_DIS
LIN {X -103.898,Y -1.308,Z -19.029,A -90.000,B 90.000,C 0.000} C_DIS
LIN {X -103.574,Y -1.308,Z -18.929,A -90.000,B 90.000,C 0.000} C_DIS
LIN {X -103.415,Y -1.308,Z -18.868,A -90.000,B 90.000,C 0.000} C_DIS
LIN {X -103.201,Y -1.308,Z -18.768,A -90.000,B 90.000,C 0.000} C_DIS
LIN {X -103.143,Y -1.308,Z -18.736,A -90.000,B 90.000,C 0.000} C_DIS
LIN {X -103.096,Y -1.308,Z -18.701,A -90.000,B 90.000,C 0.000} C_DIS
LIN {X -102.952,Y -1.308,Z -18.584,A -90.000,B 90.000,C 0.000} C_DIS
LIN {X -102.693,Y -1.308,Z -18.352,A -90.000,B 90.000,C 0.000} C_DIS
LIN {X -102.512,Y -1.308,Z -18.183,A -90.000,B 90.000,C 0.000} C_DIS
LIN {X -102.215,Y -1.308,Z -17.937,A -90.000,B 90.000,C 0.000} C_DIS
LIN {X -101.847,Y -1.308,Z -17.635,A -90.000,B 90.000,C 0.000} C_DIS
LIN {X -101.501,Y -1.308,Z -17.382,A -90.000,B 90.000,C 0.000} C_DIS
LIN {X -101.103,Y -1.308,Z -17.121,A -90.000,B 90.000,C 0.000} C_DIS
LIN {X -100.890,Y -1.308,Z -16.985,A -90.000,B 90.000,C 0.000} C_DIS
LIN {X -100.684,Y -1.308,Z -16.850,A -90.000,B 90.000,C 0.000} C_DIS
LIN {X -100.472,Y -1.308,Z -16.731,A -90.000,B 90.000,C 0.000} C_DIS
LIN {X -100.165,Y -1.308,Z -16.549,A -90.000,B 90.000,C 0.000} C_DIS
LIN {X -99.566,Y -1.308,Z -16.223,A -90.000,B 90.000,C 0.000} C_DIS
LIN {X -98.538,Y -1.308,Z -15.693,A -90.000,B 90.000,C 0.000} C_DIS
LIN {X -98.283,Y -1.308,Z -15.563,A -90.000,B 90.000,C 0.000} C_DIS
LIN {X -97.477,Y -1.308,Z -15.169,A -90.000,B 90.000,C 0.000} C_DIS
LIN {X -96.675,Y -1.308,Z -14.773,A -90.000,B 90.000,C 0.000} C_DIS
LIN {X -95.592,Y -1.308,Z -14.257,A -90.000,B 90.000,C 0.000} C_DIS
LIN {X -94.413,Y -1.308,Z -13.733,A -90.000,B 90.000,C 0.000} C_DIS
LIN {X -93.842,Y -1.308,Z -13.503,A -90.000,B 90.000,C 0.000} C_DIS
LIN {X -93.047,Y -1.308,Z -13.168,A -90.000,B 90.000,C 0.000} C_DIS
LIN {X -92.869,Y -1.308,Z -13.105,A -90.000,B 90.000,C 0.000} C_DIS
LIN {X -91.868,Y -1.308,Z -12.738,A -90.000,B 90.000,C 0.000} C_DIS
LIN {X -91.344,Y -1.308,Z -12.576,A -90.000,B 90.000,C 0.000} C_DIS
LIN {X -90.303,Y -1.308,Z -12.268,A -90.000,B 90.000,C 0.000} C_DIS
LIN {X -90.194,Y -1.308,Z -12.238,A -90.000,B 90.000,C 0.000} C_DIS
LIN {X -88.923,Y -1.308,Z -11.948,A -90.000,B 90.000,C 0.000} C_DIS
LIN {X -88.685,Y -1.308,Z -11.901,A -90.000,B 90.000,C 0.000} C_DIS
LIN {X -87.125,Y -1.308,Z -11.648,A -90.000,B 90.000,C 0.000} C_DIS
LIN {X -86.875,Y -1.308,Z -11.618,A -90.000,B 90.000,C 0.000} C_DIS
LIN {X -85.679,Y -1.308,Z -11.495,A -90.000,B 90.000,C 0.000} C_DIS
LIN {X -84.726,Y -1.308,Z -11.442,A -90.000,B 90.000,C 0.000} C_DIS
LIN {X -83.714,Y -1.308,Z -11.394,A -90.000,B 90.000,C 0.000} C_DIS
LIN {X -82.635,Y -1.308,Z -11.373,A -90.000,B 90.000,C 0.000} C_DIS
LIN {X -82.357,Y -1.308,Z -11.362,A -90.000,B 90.000,C 0.000} C_DIS
LIN {X -82.057,Y -1.308,Z -11.351,A -90.000,B 90.000,C 0.000} C_DIS
LIN {X -81.036,Y -1.308,Z -11.350,A -90.000,B 90.000,C 0.000} C_DIS
LIN {X -80.566,Y -1.308,Z -11.335,A -90.000,B 90.000,C 0.000} C_DIS
LIN {X -79.993,Y -1.308,Z -11.338,A -90.000,B 90.000,C 0.000} C_DIS
LIN {X -79.065,Y -1.308,Z -11.320,A -90.000,B 90.000,C 0.000} C_DIS
LIN {X -78.693,Y -1.308,Z -11.319,A -90.000,B 90.000,C 0.000} C_DIS
LIN {X -77.850,Y -1.308,Z -11.309,A -90.000,B 90.000,C 0.000} C_DIS
LIN {X -76.758,Y -1.308,Z -11.312,A -90.000,B 90.000,C 0.000} C_DIS
LIN {X -75.740,Y -1.308,Z -11.339,A -90.000,B 90.000,C 0.000} C_DIS
LIN {X -75.192,Y -1.308,Z -11.377,A -90.000,B 90.000,C 0.000} C_DIS
LIN {X -74.742,Y -1.308,Z -11.405,A -90.000,B 90.000,C 0.000} C_DIS
LIN {X -74.257,Y -1.308,Z -11.445,A -90.000,B 90.000,C 0.000} C_DIS
LIN {X -73.831,Y -1.308,Z -11.488,A -90.000,B 90.000,C 0.000} C_DIS
LIN {X -73.225,Y -1.308,Z -11.566,A -90.000,B 90.000,C 0.000} C_DIS
LIN {X -72.813,Y -1.308,Z -11.613,A -90.000,B 90.000,C 0.000} C_DIS
LIN {X -72.163,Y -1.308,Z -11.693,A -90.000,B 90.000,C 0.000} C_DIS
LIN {X -72.087,Y -1.308,Z -11.705,A -90.000,B 90.000,C 0.000} C_DIS
LIN {X -71.003,Y -1.308,Z -11.819,A -90.000,B 90.000,C 0.000} C_DIS
LIN {X -70.189,Y -1.308,Z -11.883,A -90.000,B 90.000,C 0.000} C_DIS
LIN {X -68.805,Y -1.308,Z -11.939,A -90.000,B 90.000,C 0.000} C_DIS
LIN {X -67.370,Y -1.308,Z -11.983,A -90.000,B 90.000,C 0.000} C_DIS
LIN {X -65.930,Y -1.308,Z -12.046,A -90.000,B 90.000,C 0.000} C_DIS
LIN {X -64.075,Y -1.308,Z -12.199,A -90.000,B 90.000,C 0.000} C_DIS
LIN {X -62.845,Y -1.308,Z -12.389,A -90.000,B 90.000,C 0.000} C_DIS
LIN {X -62.366,Y -1.308,Z -12.479,A -90.000,B 90.000,C 0.000} C_DIS
LIN {X -61.741,Y -1.308,Z -12.616,A -90.000,B 90.000,C 0.000} C_DIS
LIN {X -61.248,Y -1.308,Z -12.724,A -90.000,B 90.000,C 0.000} C_DIS
LIN {X -60.217,Y -1.308,Z -12.998,A -90.000,B 90.000,C 0.000} C_DIS
LIN {X -59.248,Y -1.308,Z -13.279,A -90.000,B 90.000,C 0.000} C_DIS
LIN {X -58.319,Y -1.308,Z -13.541,A -90.000,B 90.000,C 0.000} C_DIS
LIN {X -56.350,Y -1.308,Z -14.085,A -90.000,B 90.000,C 0.000} C_DIS
LIN {X -55.207,Y -1.308,Z -14.407,A -90.000,B 90.000,C 0.000} C_DIS
LIN {X -53.887,Y -1.308,Z -14.789,A -90.000,B 90.000,C 0.000} C_DIS
LIN {X -52.283,Y -1.308,Z -15.231,A -90.000,B 90.000,C 0.000} C_DIS
LIN {X -52.015,Y -1.308,Z -15.294,A -90.000,B 90.000,C 0.000} C_DIS
LIN {X -50.288,Y -1.308,Z -15.730,A -90.000,B 90.000,C 0.000} C_DIS
LIN {X -49.934,Y -1.308,Z -15.801,A -90.000,B 90.000,C 0.000} C_DIS
LIN {X -47.949,Y -1.308,Z -16.246,A -90.000,B 90.000,C 0.000} C_DIS
LIN {X -47.324,Y -1.308,Z -16.353,A -90.000,B 90.000,C 0.000} C_DIS
LIN {X -46.083,Y -1.308,Z -16.571,A -90.000,B 90.000,C 0.000} C_DIS
LIN {X -45.011,Y -1.308,Z -16.779,A -90.000,B 90.000,C 0.000} C_DIS
LIN {X -42.826,Y -1.308,Z -17.113,A -90.000,B 90.000,C 0.000} C_DIS
LIN {X -41.547,Y -1.308,Z -17.334,A -90.000,B 90.000,C 0.000} C_DIS
LIN {X -38.017,Y -1.308,Z -17.863,A -90.000,B 90.000,C 0.000} C_DIS
LIN {X -34.749,Y -1.308,Z -18.390,A -90.000,B 90.000,C 0.000} C_DIS
LIN {X -34.282,Y -1.308,Z -18.471,A -90.000,B 90.000,C 0.000} C_DIS
LIN {X -33.152,Y -1.308,Z -18.676,A -90.000,B 90.000,C 0.000} C_DIS
LIN {X -31.353,Y -1.308,Z -19.015,A -90.000,B 90.000,C 0.000} C_DIS
LIN {X -29.806,Y -1.308,Z -19.338,A -90.000,B 90.000,C 0.000} C_DIS
LIN {X -28.663,Y -1.308,Z -19.582,A -90.000,B 90.000,C 0.000} C_DIS
LIN {X -26.214,Y -1.308,Z -20.153,A -90.000,B 90.000,C 0.000} C_DIS
LIN {X -22.781,Y -1.308,Z -20.999,A -90.000,B 90.000,C 0.000} C_DIS
LIN {X -21.645,Y -1.308,Z -21.282,A -90.000,B 90.000,C 0.000} C_DIS
LIN {X -19.316,Y -1.308,Z -21.873,A -90.000,B 90.000,C 0.000} C_DIS
LIN {X -17.192,Y -1.308,Z -22.433,A -90.000,B 90.000,C 0.000} C_DIS
LIN {X -16.871,Y -1.308,Z -22.521,A -90.000,B 90.000,C 0.000} C_DIS
LIN {X -14.017,Y -1.308,Z -23.336,A -90.000,B 90.000,C 0.000} C_DIS
LIN {X -10.951,Y -1.308,Z -24.256,A -90.000,B 90.000,C 0.000} C_DIS
LIN {X -7.792,Y -1.308,Z -25.239,A -90.000,B 90.000,C 0.000} C_DIS
LIN {X -4.813,Y -1.308,Z -26.144,A -90.000,B 90.000,C 0.000} C_DIS
LIN {X -2.654,Y -1.308,Z -26.774,A -90.000,B 90.000,C 0.000} C_DIS
LIN {X -1.967,Y -1.308,Z -26.976,A -90.000,B 90.000,C 0.000} C_DIS
LIN {X 1.057,Y -1.308,Z -27.773,A -90.000,B 90.000,C 0.000} C_DIS
LIN {X 3.912,Y -1.308,Z -28.470,A -90.000,B 90.000,C 0.000} C_DIS
LIN {X 8.892,Y -1.308,Z -29.629,A -90.000,B 90.000,C 0.000} C_DIS
LIN {X 10.907,Y -1.308,Z -30.123,A -90.000,B 90.000,C 0.000} C_DIS
LIN {X 12.596,Y -1.308,Z -30.543,A -90.000,B 90.000,C 0.000} C_DIS
LIN {X 13.392,Y -1.308,Z -30.720,A -90.000,B 90.000,C 0.000} C_DIS
LIN {X 14.203,Y -1.308,Z -30.901,A -90.000,B 90.000,C 0.000} C_DIS
LIN {X 15.789,Y -1.308,Z -31.261,A -90.000,B 90.000,C 0.000} C_DIS
LIN {X 19.154,Y -1.308,Z -32.049,A -90.000,B 90.000,C 0.000} C_DIS
LIN {X 20.862,Y -1.308,Z -32.399,A -90.000,B 90.000,C 0.000} C_DIS
LIN {X 23.895,Y -1.308,Z -32.982,A -90.000,B 90.000,C 0.000} C_DIS
LIN {X 25.325,Y -1.308,Z -33.276,A -90.000,B 90.000,C 0.000} C_DIS
LIN {X 26.733,Y -1.308,Z -33.598,A -90.000,B 90.000,C 0.000} C_DIS
LIN {X 28.279,Y -1.308,Z -33.999,A -90.000,B 90.000,C 0.000} C_DIS
LIN {X 29.282,Y -1.308,Z -34.294,A -90.000,B 90.000,C 0.000} C_DIS
LIN {X 30.068,Y -1.308,Z -34.486,A -90.000,B 90.000,C 0.000} C_DIS
LIN {X 30.256,Y -1.308,Z -34.528,A -90.000,B 90.000,C 0.000} C_DIS
LIN {X 31.699,Y -1.308,Z -34.936,A -90.000,B 90.000,C 0.000} C_DIS
LIN {X 32.075,Y -1.308,Z -35.031,A -90.000,B 90.000,C 0.000} C_DIS
LIN {X 32.537,Y -1.308,Z -35.167,A -90.000,B 90.000,C 0.000} C_DIS
LIN {X 33.466,Y -1.308,Z -35.450,A -90.000,B 90.000,C 0.000} C_DIS
LIN {X 34.003,Y -1.308,Z -35.597,A -90.000,B 90.000,C 0.000} C_DIS
LIN {X 34.486,Y -1.308,Z -35.734,A -90.000,B 90.000,C 0.000} C_DIS
LIN {X 35.307,Y -1.308,Z -35.992,A -90.000,B 90.000,C 0.000} C_DIS
LIN {X 36.600,Y -1.308,Z -36.358,A -90.000,B 90.000,C 0.000} C_DIS
LIN {X 38.243,Y -1.308,Z -36.829,A -90.000,B 90.000,C 0.000} C_DIS
LIN {X 38.933,Y -1.308,Z -37.044,A -90.000,B 90.000,C 0.000} C_DIS
LIN {X 40.932,Y -1.308,Z -37.634,A -90.000,B 90.000,C 0.000} C_DIS
LIN {X 41.475,Y -1.308,Z -37.806,A -90.000,B 90.000,C 0.000} C_DIS
LIN {X 44.031,Y -1.308,Z -38.599,A -90.000,B 90.000,C 0.000} C_DIS
LIN {X 44.198,Y -1.308,Z -38.654,A -90.000,B 90.000,C 0.000} C_DIS
LIN {X 44.198,Y -60.000,Z -38.654,A -90.000,B 90.000,C 0.000} C_DIS

END
